METHOD objectIsValid
VAR_INPUT
	(* object which should be tested *)
	object	:CNM_AbstractObject.IObject;
	(* message if the assertion is false *)
	message	:AssertMessage;
END_VAR
IF (NOT THIS^.isObjectValid(object)) THEN
	THIS^.assertionWasWrong(message, THIS^.getDebugInfo('objectIsValid'));
END_IF
END_METHOD

(*

## Short summary
This assertion method checks if ``object``
precedes in sequence to ``objectToCompare``

.. <legal notes>

legal notes
=================
| SPDX-FileCopyrightText: © 2022 ekvip automation GmbH <info@ekvip.de>
| SPDX-License-Identifier: Apache-2.0
| For details check: Apache-2.0_

.. _Apache-2.0: https://www.apache.org/licenses/LICENSE-2.0

.. </legal notes>



*)

METHOD precedesInOrderTo
VAR_INPUT
	(* object which should be tested *)
	object			:CNM_AbstractObject.IObject;
	(* comparative object *)
	objectToCompare	:CNM_AbstractObject.IObject;
	(* message if the assertion is false *)
	message			:AssertMessage;
END_VAR
IF (THIS^.isObjectNull(THIS^.comperator)) THEN
	IF (THIS^.isObjectValid(object)) THEN
		IF (object.compareTo(objectToCompare) <> CNM_ReturnTypes.ComparationResult.SMALLER) THEN
			THIS^.assertionWasWrong(message, THIS^.getDebugInfo('precedesInOrderTo'));
		END_IF
	ELSIF (THIS^.isObjectValid(objectToCompare)) THEN
		IF (objectToCompare.compareTo(object) <= CNM_ReturnTypes.ComparationResult.EQUAL) THEN
			THIS^.assertionWasWrong(message, THIS^.getDebugInfo('precedesInOrderTo'));
		END_IF
	ELSE	
		THIS^.assertionWasWrong(message, THIS^.getDebugInfo('precedesInOrderTo'));
	END_IF
ELSIF (
	THIS^.comperator.compare(object, objectToCompare)
	<> CNM_ReturnTypes.ComparationResult.SMALLER
) THEN
	THIS^.assertionWasWrong(message, THIS^.getDebugInfo('precedesInOrderTo'));
END_IF
END_METHOD

(*

## Short summary
This allows you to set your own comperator for the methods
`IObjectAssertions.precedesInOrderTo`  
`IObjectAssertions.isEqualInOrderTo`  
`IObjectAssertions.isAfterInOrderTo`
to clear the comperator again, just call it with 0: ``foo.setComperator(comperator := 0);``

.. <legal notes>

legal notes
=================
| SPDX-FileCopyrightText: © 2022 ekvip automation GmbH <info@ekvip.de>
| SPDX-License-Identifier: Apache-2.0
| For details check: Apache-2.0_

.. _Apache-2.0: https://www.apache.org/licenses/LICENSE-2.0

.. </legal notes>



*)

METHOD setComperator
VAR_INPUT
	(* comperator to inject *)
	comperator	:CNM_AbstractObject.IComparator := 0;
END_VAR
THIS^.comperator := comperator;
END_METHOD

END_FUNCTION_BLOCK

// ---- Assertor/Assertions/PointerAssertions/classes/PointerAssertions.TcPOU
(*

## Short summary
This class provides assert statements for pointers  

.. <legal notes>

legal notes
=================
| SPDX-FileCopyrightText: © 2022 ekvip automation GmbH <info@ekvip.de>
| SPDX-License-Identifier: Apache-2.0
| For details check: Apache-2.0_

.. _Apache-2.0: https://www.apache.org/licenses/LICENSE-2.0

.. </legal notes>



*)

{attribute 'reflection'}
FUNCTION_BLOCK PointerAssertions EXTENDS AbstractAssertion IMPLEMENTS IPointerAssertions
VAR
END_VAR

(*

## Short summary
This abstract property returns the class name of the concrete object, 
It's for debugging purpose

.. <legal notes>

legal notes
=================
| SPDX-FileCopyrightText: © 2022 ekvip automation GmbH <info@ekvip.de>
| SPDX-License-Identifier: Apache-2.0
| For details check: Apache-2.0_

.. _Apache-2.0: https://www.apache.org/licenses/LICENSE-2.0

.. </legal notes>

*)

PROPERTY className :CNM_AbstractObject.ClassName
GET
className := 'CNM_Assertor.PointerAssertions';
END_GET
END_PROPERTY

(*

## Short summary
This assertion method checks if pointer is aligned with register size.

.. <legal notes>

legal notes
=================
| SPDX-FileCopyrightText: © 2025 ekvip automation GmbH <info@ekvip.de>
| SPDX-License-Identifier: Apache-2.0
| For details check: Apache-2.0_

.. _Apache-2.0: https://www.apache.org/licenses/LICENSE-2.0

.. </legal notes>



*)

METHOD isAligned
VAR_INPUT
	(* memory address *)
	address		:PVOID;
	(* message if the assertion is false *)
	message		:AssertMessage;
END_VAR
VAR CONSTANT
	SIZE :PVOID := SIZEOF(__XWORD);
END_VAR
IF (address MOD SIZE > 0) THEN
	THIS^.assertionWasWrong(message, THIS^.getDebugInfo('isAligned'));
END_IF
END_METHOD

(*

## Short summary
This assertion method checks if pointer is aligned with DWord size.

.. <legal notes>

legal notes
=================
| SPDX-FileCopyrightText: © 2025 ekvip automation GmbH <info@ekvip.de>
| SPDX-License-Identifier: Apache-2.0
| For details check: Apache-2.0_

.. _Apache-2.0: https://www.apache.org/licenses/LICENSE-2.0

.. </legal notes>



*)

METHOD isDwordAligned
VAR_INPUT
	(* memory address *)
	address		:PVOID;
	(* message if the assertion is false *)
	message		:AssertMessage;
END_VAR
VAR CONSTANT
	SIZE :PVOID := SIZEOF(DWORD);
END_VAR
IF (address MOD SIZE > 0) THEN
	THIS^.assertionWasWrong(message, THIS^.getDebugInfo('isAligned'));
END_IF
END_METHOD

(*

## Short summary
This assertion method checks if ``address1`` and ``address2`` refer to the same address

.. <legal notes>

legal notes
=================
| SPDX-FileCopyrightText: © 2022 ekvip automation GmbH <info@ekvip.de>
| SPDX-License-Identifier: Apache-2.0
| For details check: Apache-2.0_

.. _Apache-2.0: https://www.apache.org/licenses/LICENSE-2.0

.. </legal notes>



*)

METHOD isEqualTo
VAR_INPUT
	(* memory address *)
	address1	:PVOID;
	(* memory address *)
	address2	:PVOID;
	(* message if the assertion is false *)
	message		:AssertMessage;
END_VAR
IF (address1 <> address2) THEN
	THIS^.assertionWasWrong(message, THIS^.getDebugInfo('isEqualTo'));
END_IF
END_METHOD

(*

## Short summary
This assertion method checks if pointer is aligned with Lword size.

.. <legal notes>

legal notes
=================
| SPDX-FileCopyrightText: © 2025 ekvip automation GmbH <info@ekvip.de>
| SPDX-License-Identifier: Apache-2.0
| For details check: Apache-2.0_

.. _Apache-2.0: https://www.apache.org/licenses/LICENSE-2.0

.. </legal notes>



*)

METHOD isLwordAligned
VAR_INPUT
	(* memory address *)
	address		:PVOID;
	(* message if the assertion is false *)
	message		:AssertMessage;
END_VAR
VAR CONSTANT
	SIZE :PVOID := SIZEOF(LWORD);
END_VAR
IF (address MOD SIZE > 0) THEN
	THIS^.assertionWasWrong(message, THIS^.getDebugInfo('isAligned'));
END_IF
END_METHOD

(*

## Short summary
This assertion method checks if ``address1`` and ``address2`` refer not to the same address

.. <legal notes>

legal notes
=================
| SPDX-FileCopyrightText: © 2022 ekvip automation GmbH <info@ekvip.de>
| SPDX-License-Identifier: Apache-2.0
| For details check: Apache-2.0_

.. _Apache-2.0: https://www.apache.org/licenses/LICENSE-2.0

.. </legal notes>



*)

METHOD isNotEqualTo
VAR_INPUT
	(* memory address *)
	address1	:PVOID;
	(* memory address *)
	address2	:PVOID;
	(* message if the assertion is false *)
	message		:AssertMessage;
END_VAR
IF (address1 = address2) THEN
	THIS^.assertionWasWrong(message, THIS^.getDebugInfo('isNotEqualTo'));
END_IF
END_METHOD

(*

## Short summary
This assertion method checks if pointer is not null

.. <legal notes>

legal notes
=================
| SPDX-FileCopyrightText: © 2022 ekvip automation GmbH <info@ekvip.de>
| SPDX-License-Identifier: Apache-2.0
| For details check: Apache-2.0_

.. _Apache-2.0: https://www.apache.org/licenses/LICENSE-2.0

.. </legal notes>



*)

METHOD isNotNull
VAR_INPUT
	(* memory address *)
	address	:PVOID;
	(* message if the assertion is false *)
	message	:AssertMessage;
END_VAR
IF (address = 0) THEN
	THIS^.assertionWasWrong(message, THIS^.getDebugInfo('isNotNull'));
END_IF
END_METHOD

(*

## Short summary
This assertion method checks if memory areas are overlapping

.. <legal notes>

legal notes
=================
| SPDX-FileCopyrightText: © 2022 ekvip automation GmbH <info@ekvip.de>
| SPDX-License-Identifier: Apache-2.0
| For details check: Apache-2.0_

.. _Apache-2.0: https://www.apache.org/licenses/LICENSE-2.0

.. </legal notes>



*)

METHOD isNotOverlapping
VAR_INPUT
	(* memory address *)
	address1	:PVOID;
	(* memory address *)
	address2	:PVOID;
	(*the size of the memory area identified by address1*)
	sizeInBytes1		:UDINT;
	(*the size of the memory area identified by address2*)
	sizeInBytes2		:UDINT;
	(* message if the assertion is false *)
	message		:AssertMessage;
END_VAR
IF 	(( 
		address1 = address2
	) OR_ELSE(
		//address1 + sizeInBytes1 < address1 is to protect overflows caused by the calculation address1 + sizeInBytes1
		(address1 < address2) AND_THEN ((address1 + sizeInBytes1 < address1) OR_ELSE ((address1 + sizeInBytes1) >= address2))
	) OR_ELSE (
		//address2 + sizeInBytes2 < address2 is to protect overflows caused by the calculation address2 + sizeInBytes2
		(address1 > address2) AND_THEN (((address2 + sizeInBytes2 < address2) OR_ELSE ((address2 + sizeInBytes2) >= address1)))
	)
) THEN
		THIS^.assertionWasWrong(message, THIS^.getDebugInfo('isNotOverlapping'));
END_IF
END_METHOD

(*

## Short summary
This assertion method checks if pointer is null

.. <legal notes>

legal notes
=================
| SPDX-FileCopyrightText: © 2022 ekvip automation GmbH <info@ekvip.de>
| SPDX-License-Identifier: Apache-2.0
| For details check: Apache-2.0_

.. _Apache-2.0: https://www.apache.org/licenses/LICENSE-2.0

.. </legal notes>



*)

METHOD isNull
VAR_INPUT
	(* memory address *)
	address	:PVOID;
	(* message if the assertion is false *)
	message	:AssertMessage;
END_VAR
IF (address <> 0) THEN
	THIS^.assertionWasWrong(message, THIS^.getDebugInfo('isNull'));
END_IF
END_METHOD

(*

## Short summary
This assertion method checks if memory areas are overlapping

.. <legal notes>

legal notes
=================
| SPDX-FileCopyrightText: © 2022 ekvip automation GmbH <info@ekvip.de>
| SPDX-License-Identifier: Apache-2.0
| For details check: Apache-2.0_

.. _Apache-2.0: https://www.apache.org/licenses/LICENSE-2.0

.. </legal notes>



*)

METHOD isOverlapping
VAR_INPUT
	(* memory address *)
	address1	:PVOID;
	(* memory address *)
	address2	:PVOID;
	(*the size of the memory area identified by address1*)
	sizeInBytes1		:UDINT;
	(*the size of the memory area identified by address2*)
	sizeInBytes2		:UDINT;
	(* message if the assertion is false *)
	message		:AssertMessage;
END_VAR
RETURN(address1 = address2);
IF ((
		(address1 < address2) AND_THEN ((address1 + sizeInBytes1) < address2)
	) OR_ELSE (
		(address1 > address2) AND_THEN ((address2 + sizeInBytes2) < address1)
	)
) THEN
	THIS^.assertionWasWrong(message, THIS^.getDebugInfo('isOverlapping'));
END_IF;
END_METHOD

(*

## Short summary
This assertion method checks if pointer is valid.
That means the pointer and size are not zero,
the pointer is in a valid area.

**Attention:** 
	Validity of the pointer will be proofed for 32 bit systems only.
	For other systems it's an optimistic estimate.

.. <legal notes>

legal notes
=================
| SPDX-FileCopyrightText: © 2022 ekvip automation GmbH <info@ekvip.de>
| SPDX-License-Identifier: Apache-2.0
| For details check: Apache-2.0_

.. _Apache-2.0: https://www.apache.org/licenses/LICENSE-2.0

.. </legal notes>



*)

METHOD isValid
VAR_INPUT
	(* memory address *)
	address		:PVOID;
	(* number of bytes *)
	sizeInBytes	:UDINT;
	(* message if the assertion is false *)
	message		:AssertMessage;
END_VAR
VAR
	{attribute 'displaymode':='hex'}
	stackAddress	:__XWORD;
	testPointer		:POINTER TO BYTE := NULL;
	testByte		:BYTE;
	exc				: __SYSTEM.ExceptionCode;
END_VAR
VAR CONSTANT
	{attribute 'displaymode':='hex'}
	NULL :__XWORD := 0;
	{attribute 'displaymode':='hex'}
	REGISTER_SIZE :UDINT := SIZEOF(__XWORD);
	(* 0x400000 is 4096kb and this is the max configurable stack size *)
	{attribute 'displaymode':='hex'}
	MAX_STACK_SIZE :__XWORD := 16#0040_0000;
END_VAR
stackAddress := ADR(stackAddress);
IF (
	(address = NULL) 
	OR_ELSE (sizeInBytes = NULL)
	//check for overflow
	OR_ELSE (address + sizeInBytes < address)
	OR_ELSE (
		(Tc2_System.F_CheckMemoryArea(pData := address, nSize := sizeInBytes) = Tc2_System.E_TcMemoryArea.Unknown)
		AND_THEN (address < ABS(stackAddress - MAX_STACK_SIZE))
	)
) THEN
	THIS^.assertionWasWrong(message, THIS^.getDebugInfo('isValid'));
ELSE
	testPointer := address;
	__TRY
		testByte := testPointer^;
	__CATCH(exc)
		THIS^.assertionWasWrong(message, THIS^.getDebugInfo('isValid'));
	__ENDTRY
END_IF
END_METHOD

(*

## Short summary
This assertion method checks if pointer is aligned with word size.

.. <legal notes>

legal notes
=================
| SPDX-FileCopyrightText: © 2025 ekvip automation GmbH <info@ekvip.de>
| SPDX-License-Identifier: Apache-2.0
| For details check: Apache-2.0_

.. _Apache-2.0: https://www.apache.org/licenses/LICENSE-2.0

.. </legal notes>



*)

METHOD isWordAligned
VAR_INPUT
	(* memory address *)
	address		:PVOID;
	(* message if the assertion is false *)
	message		:AssertMessage;
END_VAR
VAR CONSTANT
	SIZE :PVOID := SIZEOF(WORD);
END_VAR
IF (address MOD SIZE > 0) THEN
	THIS^.assertionWasWrong(message, THIS^.getDebugInfo('isAligned'));
END_IF
END_METHOD

(*

## Short summary
This assertion method checks if pointer refers to cnc area

.. <legal notes>

legal notes
=================
| SPDX-FileCopyrightText: © 2022 ekvip automation GmbH <info@ekvip.de>
| SPDX-License-Identifier: Apache-2.0
| For details check: Apache-2.0_

.. _Apache-2.0: https://www.apache.org/licenses/LICENSE-2.0

.. </legal notes>



*)

METHOD memoryAreaIsCnc
VAR_INPUT
	(* memory address *)
	address		:PVOID;
	(* number of bytes *)
	sizeInBytes	:UDINT;
	(* message if the assertion is false *)
	message		:AssertMessage;
END_VAR
IF (
	Tc2_System.F_CheckMemoryArea(
		pData := address,
		nSize := sizeInBytes
	) <> Tc2_System.E_TcMemoryArea.CNC
) THEN
	THIS^.assertionWasWrong(message, THIS^.getDebugInfo('memoryAreaIsCnc'));
END_IF
END_METHOD

(*

## Short summary
This assertion method checks if pointer refers to dynamic area

.. <legal notes>

legal notes
=================
| SPDX-FileCopyrightText: © 2022 ekvip automation GmbH <info@ekvip.de>
| SPDX-License-Identifier: Apache-2.0
| For details check: Apache-2.0_

.. _Apache-2.0: https://www.apache.org/licenses/LICENSE-2.0

.. </legal notes>



*)

METHOD memoryAreaIsDynamic
VAR_INPUT
	(* memory address *)
	address		:PVOID;
	(* number of bytes *)
	sizeInBytes	:UDINT;
	(* message if the assertion is false *)
	message		:AssertMessage;
END_VAR
IF (
	Tc2_System.F_CheckMemoryArea(
		pData := address,
		nSize := sizeInBytes
	) <> Tc2_System.E_TcMemoryArea.Dynamic
) THEN
	THIS^.assertionWasWrong(message, THIS^.getDebugInfo('memoryAreaIsDynamic'));
END_IF
END_METHOD

(*

## Short summary
This assertion method checks if pointer refers not to cnc area

.. <legal notes>

legal notes
=================
| SPDX-FileCopyrightText: © 2022 ekvip automation GmbH <info@ekvip.de>
| SPDX-License-Identifier: Apache-2.0
| For details check: Apache-2.0_

.. _Apache-2.0: https://www.apache.org/licenses/LICENSE-2.0

.. </legal notes>



*)

METHOD memoryAreaIsNotCnc
VAR_INPUT
	(* memory address *)
	address		:PVOID;
	(* number of bytes *)
	sizeInBytes	:UDINT;
	(* message if the assertion is false *)
	message		:AssertMessage;
END_VAR
IF (
	Tc2_System.F_CheckMemoryArea(
		pData := address,
		nSize := sizeInBytes
	) = Tc2_System.E_TcMemoryArea.CNC
) THEN
	THIS^.assertionWasWrong(message, THIS^.getDebugInfo('memoryAreaIsNotCnc'));
END_IF
END_METHOD

(*

## Short summary
This assertion method checks if pointer refers not to dynamic area

.. <legal notes>

legal notes
=================
| SPDX-FileCopyrightText: © 2022 ekvip automation GmbH <info@ekvip.de>
| SPDX-License-Identifier: Apache-2.0
| For details check: Apache-2.0_

.. _Apache-2.0: https://www.apache.org/licenses/LICENSE-2.0

.. </legal notes>



*)

METHOD memoryAreaIsNotDynamic
VAR_INPUT
	(* memory address *)
	address		:PVOID;
	(* number of bytes *)
	sizeInBytes	:UDINT;
	(* message if the assertion is false *)
	message		:AssertMessage;
END_VAR
IF (
	Tc2_System.F_CheckMemoryArea(
		pData := address,
		nSize := sizeInBytes
	) = Tc2_System.E_TcMemoryArea.Dynamic
) THEN
	THIS^.assertionWasWrong(message, THIS^.getDebugInfo('memoryAreaIsNotDynamic'));
END_IF
END_METHOD

(*

## Short summary
This assertion method checks if pointer refers not to static area

.. <legal notes>

legal notes
=================
| SPDX-FileCopyrightText: © 2022 ekvip automation GmbH <info@ekvip.de>
| SPDX-License-Identifier: Apache-2.0
| For details check: Apache-2.0_

.. _Apache-2.0: https://www.apache.org/licenses/LICENSE-2.0

.. </legal notes>



*)

METHOD memoryAreaIsNotStatic
VAR_INPUT
	(* memory address *)
	address		:PVOID;
	(* number of bytes *)
	sizeInBytes	:UDINT;
	(* message if the assertion is false *)
	message		:AssertMessage;
END_VAR
IF (
	Tc2_System.F_CheckMemoryArea(
		pData := address,
		nSize := sizeInBytes
	) = Tc2_System.E_TcMemoryArea.Static
) THEN
	THIS^.assertionWasWrong(message, THIS^.getDebugInfo('memoryAreaIsNotStatic'));
END_IF
END_METHOD

(*

## Short summary
This assertion method checks if pointer is not at memory area unknown

.. <legal notes>

legal notes
=================
| SPDX-FileCopyrightText: © 2022 ekvip automation GmbH <info@ekvip.de>
| SPDX-License-Identifier: Apache-2.0
| For details check: Apache-2.0_

.. _Apache-2.0: https://www.apache.org/licenses/LICENSE-2.0

.. </legal notes>



*)

METHOD memoryAreaIsNotUnkown
VAR_INPUT
	(* memory address *)
	address		:PVOID;
	(* number of bytes *)
	sizeInBytes	:UDINT;
	(* message if the assertion is false *)
	message		:AssertMessage;
END_VAR
IF (
	Tc2_System.F_CheckMemoryArea(
		pData := address,
		nSize := sizeInBytes
	) = Tc2_System.E_TcMemoryArea.Unknown
) THEN
	THIS^.assertionWasWrong(message, THIS^.getDebugInfo('memoryAreaIsNotUnkown'));
END_IF
END_METHOD

(*

## Short summary
This assertion method checks if pointer refers to static area

.. <legal notes>

legal notes
=================
| SPDX-FileCopyrightText: © 2022 ekvip automation GmbH <info@ekvip.de>
| SPDX-License-Identifier: Apache-2.0
| For details check: Apache-2.0_

.. _Apache-2.0: https://www.apache.org/licenses/LICENSE-2.0

.. </legal notes>



*)

METHOD memoryAreaIsStatic
VAR_INPUT
	(* memory address *)
	address		:PVOID;
	(* number of bytes *)
	sizeInBytes	:UDINT;
	(* message if the assertion is false *)
	message		:AssertMessage;
END_VAR
IF (
	Tc2_System.F_CheckMemoryArea(
		pData := address,
		nSize := sizeInBytes
	) <> Tc2_System.E_TcMemoryArea.Static
) THEN
	THIS^.assertionWasWrong(message, THIS^.getDebugInfo('memoryAreaIsStatic'));
END_IF
END_METHOD

(*

## Short summary
This assertion method checks if pointer refers not to an unknown area

.. <legal notes>

legal notes
=================
| SPDX-FileCopyrightText: © 2022 ekvip automation GmbH <info@ekvip.de>
| SPDX-License-Identifier: Apache-2.0
| For details check: Apache-2.0_

.. _Apache-2.0: https://www.apache.org/licenses/LICENSE-2.0

.. </legal notes>



*)

METHOD memoryAreaIsUnkown
VAR_INPUT
	(* memory address *)
	address		:PVOID;
	(* number of bytes *)
	sizeInBytes	:UDINT;
	(* message if the assertion is false *)
	message		:AssertMessage;
END_VAR
IF (
	Tc2_System.F_CheckMemoryArea(
		pData := address,
		nSize := sizeInBytes
	) <> Tc2_System.E_TcMemoryArea.Unknown
) THEN
	THIS^.assertionWasWrong(message, THIS^.getDebugInfo('memoryAreaIsUnkown'));
END_IF
END_METHOD

END_FUNCTION_BLOCK

// ---- Assertor/Assertions/StringAssertion/classes/StringAssertions.TcPOU
(*

## Short summary

This class provides assert statements for strings
For UTF-16 strings up to 255 ``WORD`` (``WSTRING(Tc2_System.MAX_STRING_LENGTH)``) use the property `IStringAssertions.utf16`.
For windows-1252 strings up to 255 ``BYTE`` (``Tc2_System.T_MaxString``) use the property `IStringAssertions.windows1252`.
For windows-1252 or UTF-16 strings that are longer, use the property `IStringAssertions.anyString`  

.. <legal notes>

legal notes
=================
| SPDX-FileCopyrightText: © 2022 ekvip automation GmbH <info@ekvip.de>
| SPDX-License-Identifier: Apache-2.0
| For details check: Apache-2.0_

.. _Apache-2.0: https://www.apache.org/licenses/LICENSE-2.0

.. </legal notes>



*)

{attribute 'reflection'}
FUNCTION_BLOCK INTERNAL StringAssertions EXTENDS CNM_AbstractObject.Object IMPLEMENTS IStringAssertions, IAssertCallBackSetter
VAR
	(* class to handle windows-1252 and windows-1251 assertions *)
	win125xStringAssertions	:Windows125xStringAssertions();
	(* class to handle UTF-16 assertions *)
	utf16StringAssertions	:Utf16StringAssertions();
	(* class to handle UTF-8 assertions *)
	utf8StringAssertions	:Utf8StringAssertions();
	(* class to handle Unicode assertions with anys string*)
	UnicodeAssertions :UnicodeAssertions();
END_VAR

(*

## Short summary
This abstract property returns the class name of the concrete object, 
It's for debugging purpose

.. <legal notes>

legal notes
=================
| SPDX-FileCopyrightText: © 2022 ekvip automation GmbH <info@ekvip.de>
| SPDX-License-Identifier: Apache-2.0
| For details check: Apache-2.0_

.. _Apache-2.0: https://www.apache.org/licenses/LICENSE-2.0

.. </legal notes>

*)

PROPERTY className :CNM_AbstractObject.ClassName
GET
className := 'CNM_Assertor.StringAssertions';
END_GET
END_PROPERTY

(*

## Short summary
This methods is the setter for the callback class if an assertion was false

.. <legal notes>

legal notes
=================
| SPDX-FileCopyrightText: © 2022 ekvip automation GmbH <info@ekvip.de>
| SPDX-License-Identifier: Apache-2.0
| For details check: Apache-2.0_

.. _Apache-2.0: https://www.apache.org/licenses/LICENSE-2.0

.. </legal notes>



*)

METHOD setCallBack
VAR_INPUT
	(* the class that must be informed if an assertion is false *)
	callBack	: IAssertCallBack;
END_VAR
THIS^.utf16StringAssertions.setCallBack(callBack);
THIS^.win125xStringAssertions.setCallBack(callBack);
THIS^.utf8StringAssertions.setCallBack(callBack);
THIS^.UnicodeAssertions.setCallBack(callBack);
END_METHOD

(*

## Short summary
Returns an interface `IUnicodeStringAssertions` with assert statements,
for UTF-8 and UTF-16 strings with an undefined length.

**Attention:** 
	All strings are handled as null terminated byte/word streams.
	For UTF-8 is end of the string 16#00
	For UTF-16 is end of the string 16#00_00

**Attention:** 
	The interface `IUnicodeAssertions` uses ``ANY_STRING``, 
	for this it's not possible to use literals/constants,
	because for ``ANY`` types generates the compiler ``__SYSTEM.AnyType``
	and ``__SYSTEM.AnyType`` contains a pointer  

.. <legal notes>

legal notes
=================
| SPDX-FileCopyrightText: © 2022 ekvip automation GmbH <info@ekvip.de>
| SPDX-License-Identifier: Apache-2.0
| For details check: Apache-2.0_

.. _Apache-2.0: https://www.apache.org/licenses/LICENSE-2.0

.. </legal notes>

*)
PROPERTY unicode :IUnicodeStringAssertions
GET
unicode := THIS^.UnicodeAssertions;
END_GET
END_PROPERTY

(*

## Short summary
Returns an interface `IUtf16StringAssertions` with assert statements
for UTF-16 strings until 255 ``WORD`` length (``WSTRING(Tc2_System.MAX_STRING_LENGTH)``)

.. <legal notes>

legal notes
=================
| SPDX-FileCopyrightText: © 2022 ekvip automation GmbH <info@ekvip.de>
| SPDX-License-Identifier: Apache-2.0
| For details check: Apache-2.0_

.. _Apache-2.0: https://www.apache.org/licenses/LICENSE-2.0

.. </legal notes>

*)

PROPERTY utf16 :IUtf16StringAssertions
GET
utf16 := THIS^.utf16StringAssertions;
END_GET
END_PROPERTY

(*

## Short summary
Returns an interface `IUtf8StringAssertions` with assert statements
for UTF-8 strings up to 255 bytes length (``STRING(Tc2_System.MAX_STRING_LENGTH)``)

.. <legal notes>

legal notes
=================
| SPDX-FileCopyrightText: © 2022 ekvip automation GmbH <info@ekvip.de>
| SPDX-License-Identifier: Apache-2.0
| For details check: Apache-2.0_

.. _Apache-2.0: https://www.apache.org/licenses/LICENSE-2.0

.. </legal notes>

*)

PROPERTY utf8 :IUtf8StringAssertions
GET
utf8 := THIS^.utf8StringAssertions;
END_GET
END_PROPERTY

(*

## Short summary
Returns an interface `IWindows125xStringAssertions` with assert statements for 8-bit 
windows-1252 and windows-1251 strings up to 255 characters length (``Tc2_System.T_MaxString``).
Use Tc2_Utilities.GLOBAL_SBCS_TABLE variable to select required encoding

.. <legal notes>

legal notes
=================
| SPDX-FileCopyrightText: © 2022 ekvip automation GmbH <info@ekvip.de>
| SPDX-License-Identifier: Apache-2.0
| For details check: Apache-2.0_

.. _Apache-2.0: https://www.apache.org/licenses/LICENSE-2.0

.. </legal notes>

*)

PROPERTY windows125x :IWindows125xStringAssertions
GET
windows125x := THIS^.win125xStringAssertions;
END_GET
END_PROPERTY

END_FUNCTION_BLOCK

// ---- Assertor/Assertions/StringAssertion/Win125x/classes/Windows125xStringAssertions.TcPOU
(*

## Short summary
This class provides assert statements for Windows-1252 and Windows-1251 strings up to 255 characters length. 
Used encoding is specified in ``Tc2_Utilities.GLOBAL_SBCS_TABLE`` global variable

**Attention:** 
	All strings are handled as null-terminated byte streams

.. <legal notes>

legal notes
=================
| SPDX-FileCopyrightText: © 2024 ekvip automation GmbH <info@ekvip.de>
| SPDX-License-Identifier: Apache-2.0
| For details check: Apache-2.0_

.. _Apache-2.0: https://www.apache.org/licenses/LICENSE-2.0

.. </legal notes>



*)

{attribute 'reflection'}
FUNCTION_BLOCK INTERNAL Windows125xStringAssertions EXTENDS AbstractAssertion IMPLEMENTS IWindows125xStringAssertions
VAR
	(* class to handle the windows-1252 and windows-1251 string assertions *)  
	assertion	:Windows125xStringPointerAssertions();
END_VAR

(*

## Short summary
This abstract property returns the class name of the concrete object, 
It's for debugging purpose

.. <legal notes>

legal notes
=================
| SPDX-FileCopyrightText: © 2022 ekvip automation GmbH <info@ekvip.de>
| SPDX-License-Identifier: Apache-2.0
| For details check: Apache-2.0_

.. _Apache-2.0: https://www.apache.org/licenses/LICENSE-2.0

.. </legal notes>

*)

PROPERTY className :CNM_AbstractObject.ClassName
GET
className := 'CNM_Assertor.Windows125xStringAssertions';
END_GET
END_PROPERTY

(*

## Short summary
This assertion method checks if the current string ``stringToCheck`` contains the search string ``searchString``.
Processed strings must be in UTF-8 encoding

.. <legal notes>

legal notes
=================
| SPDX-FileCopyrightText: © 2024 ekvip automation GmbH <info@ekvip.de>
| SPDX-License-Identifier: Apache-2.0
| For details check: Apache-2.0_

.. _Apache-2.0: https://www.apache.org/licenses/LICENSE-2.0

.. </legal notes>



*)

METHOD contains
VAR_INPUT
	(* current string to check *)
	stringToCheck	:Tc2_System.T_MaxString;
	(* string must be found in ``stringToCheck`` *)
	searchString	:Tc2_System.T_MaxString;
	(* message if the assertion is false *)
	message			:AssertMessage;
	(* used Single Byte Character Set (SBCS), is set in Tc2_Utilities.GLOBAL_SBCS_TABLE *)
	sbcsType 		:Tc2_Utilities.E_SBCSType := Tc2_Utilities.E_SBCSType.eSBCS_WesternEuropean;
	(* ``TRUE`` means ignore cases; ``FALSE`` means that cases must be equal too *)
	ignoreCases		:BOOL := FALSE;
END_VAR
assertion.contains(
	stringToCheck 	:= ADR(stringToCheck),
	searchString  	:= ADR(searchString),
	ignoreCases 	:= ignoreCases,
	message 		:= message,
	sbcsType 		:= sbcsType
);
END_METHOD

(*

## Short summary
This assertion method checks if the current string ``stringToCheck`` doesn't contain the search string ``searchString``.
Processed strings must be in UTF-8 encoding

.. <legal notes>

legal notes
=================
| SPDX-FileCopyrightText: © 2024 ekvip automation GmbH <info@ekvip.de>
| SPDX-License-Identifier: Apache-2.0
| For details check: Apache-2.0_

.. _Apache-2.0: https://www.apache.org/licenses/LICENSE-2.0

.. </legal notes>



*)

METHOD containsNo
VAR_INPUT
	(* current string to check *)
	stringToCheck	:Tc2_System.T_MaxString;
	(* string that must not be found in ``stringToCheck`` *)
	searchString	:Tc2_System.T_MaxString;
	(* message if the assertion is false *)
	message			:AssertMessage;
	(* used Single Byte Character Set (SBCS), is set in Tc2_Utilities.GLOBAL_SBCS_TABLE *)
	sbcsType 		:Tc2_Utilities.E_SBCSType := Tc2_Utilities.E_SBCSType.eSBCS_WesternEuropean;
	(* ``TRUE`` means ignore cases; ``FALSE`` means that cases must be equal too *)
	ignoreCases		:BOOL := FALSE;
END_VAR
THIS^.assertion.containsNo(
	stringToCheck 	:= ADR(stringToCheck),
	searchString 	:= ADR(searchString),
	ignoreCases 	:= ignoreCases,
	message 		:= message,
	sbcsType 		:= sbcsType
);
END_METHOD

(*

## Short summary
This assertion method checks if the current string ``stringToCheck`` ends with the string ``end``.
Processed strings must be in UTF-8 encoding

.. <legal notes>

legal notes
=================
| SPDX-FileCopyrightText: © 2024 ekvip automation GmbH <info@ekvip.de>
| SPDX-License-Identifier: Apache-2.0
| For details check: Apache-2.0_

.. _Apache-2.0: https://www.apache.org/licenses/LICENSE-2.0

.. </legal notes>



*)

METHOD endsWith
VAR_INPUT
	(* current string to check *)
	stringToCheck	:Tc2_System.T_MaxString;
	(* expected end of ``stringToCheck`` *)
	end				:Tc2_System.T_MaxString;
	(* message if the assertion is false *)
	message			:AssertMessage;
	(* used Single Byte Character Set (SBCS), is set in Tc2_Utilities.GLOBAL_SBCS_TABLE *)
	sbcsType 		:Tc2_Utilities.E_SBCSType := Tc2_Utilities.E_SBCSType.eSBCS_WesternEuropean;
	(* ``TRUE`` means ignore cases; ``FALSE`` means that cases must be equal too *)
	ignoreCases		:BOOL := FALSE;
	(* ``TRUE`` means truncation of spaces on the right side of ``stringToCheck``*)
	trim		:BOOL := FALSE;
END_VAR
assertion.endsWith(
	stringToCheck	:= ADR(stringToCheck),
	end				:= ADR(end),
	ignoreCases		:= ignoreCases,
	trim			:= trim,
	message			:= message,
	sbcsType 		:= sbcsType
);
END_METHOD

(*

## Short summary
This assertion method checks if the current string ``stringToCheck`` is empty.
Processed strings must be in UTF-8 encoding

.. <legal notes>

legal notes
=================
| SPDX-FileCopyrightText: © 2024 ekvip automation GmbH <info@ekvip.de>
| SPDX-License-Identifier: Apache-2.0
| For details check: Apache-2.0_

.. _Apache-2.0: https://www.apache.org/licenses/LICENSE-2.0

.. </legal notes>



*)

METHOD isEmpty
VAR_INPUT
	(* current string to check *)
	stringToCheck	:Tc2_System.T_MaxString;
	(* message if the assertion is false *)
	message			:AssertMessage;
END_VAR
IF (stringToCheck <> '') THEN
	THIS^.assertionWasWrong(message, THIS^.getDebugInfo('isEmpty'));
END_IF
END_METHOD

(*

## Short summary
This assertion method checks if the current string ``stringToCheck`` is equal to ``expected``.
Processed strings must be in UTF-8 encoding

.. <legal notes>

legal notes
=================
| SPDX-FileCopyrightText: © 2024 ekvip automation GmbH <info@ekvip.de>
| SPDX-License-Identifier: Apache-2.0
| For details check: Apache-2.0_

.. _Apache-2.0: https://www.apache.org/licenses/LICENSE-2.0

.. </legal notes>



*)

METHOD isEqualTo
VAR_INPUT
	(* current string to check *)
	stringToCheck	:Tc2_System.T_MaxString;
	(* ``stringToCheck`` must be equal to expected *)
	expected		:Tc2_System.T_MaxString;
	(* message if the assertion is false *)
	message			:AssertMessage;
	(* used Single Byte Character Set (SBCS), is set in Tc2_Utilities.GLOBAL_SBCS_TABLE *)
	sbcsType 		:Tc2_Utilities.E_SBCSType := Tc2_Utilities.E_SBCSType.eSBCS_WesternEuropean;
	(* ``TRUE`` means ignore cases; ``FALSE`` means that cases must be equal too *)
	ignoreCases		:BOOL := FALSE;
END_VAR
assertion.isEqualTo(
	stringToCheck	:= ADR(stringToCheck),
	expected		:= ADR(expected),
	ignoreCases		:= ignoreCases,
	message			:= message,
	sbcsType 		:= sbcsType
);
END_METHOD

(*

## Short summary
This assertion method checks if the current string ``stringToCheck`` is not empty.
Processed strings must be in UTF-8 encoding

.. <legal notes>

legal notes
=================
| SPDX-FileCopyrightText: © 2024 ekvip automation GmbH <info@ekvip.de>
| SPDX-License-Identifier: Apache-2.0
| For details check: Apache-2.0_

.. _Apache-2.0: https://www.apache.org/licenses/LICENSE-2.0

.. </legal notes>



*)

METHOD isNotEmpty
VAR_INPUT
	(* current string to check *)
	stringToCheck	:Tc2_System.T_MaxString;
	(* message if the assertion is false *)
	message			:AssertMessage;
END_VAR
IF (stringToCheck = '') THEN
	THIS^.assertionWasWrong(message, THIS^.getDebugInfo('isEmpty'));
END_IF
END_METHOD

(*

## Short summary
This assertion method checks if the current string ``stringToCheck`` is not equal to ``unexpected``.
Processed strings must be in UTF-8 encoding

.. <legal notes>

legal notes
=================
| SPDX-FileCopyrightText: © 2024 ekvip automation GmbH <info@ekvip.de>
| SPDX-License-Identifier: Apache-2.0
| For details check: Apache-2.0_

.. _Apache-2.0: https://www.apache.org/licenses/LICENSE-2.0

.. </legal notes>



*)

METHOD isNotEqualTo
VAR_INPUT
	(* current string to check *)
	stringToCheck	:Tc2_System.T_MaxString;
	(* ``stringToCheck`` must be not equal to expected *)
	unexpected		:Tc2_System.T_MaxString;
	(* message if the assertion is false *)
	message			:AssertMessage;
	(* used Single Byte Character Set (SBCS), is set in Tc2_Utilities.GLOBAL_SBCS_TABLE *)
	sbcsType 		:Tc2_Utilities.E_SBCSType := Tc2_Utilities.E_SBCSType.eSBCS_WesternEuropean;
	(* ``TRUE`` means ignore cases; ``FALSE`` means that cases must be equal too *)
	ignoreCases		:BOOL := FALSE;
END_VAR
THIS^.assertion.isNotEqualTo(
	stringToCheck	:= ADR(stringToCheck),
	unexpected		:= ADR(unexpected),
	ignoreCases		:= ignoreCases,
	message			:= message,
	sbcsType 		:= sbcsType
);
END_METHOD

(*

## Short summary
This assertion method checks if the current string ``stringToCheck`` length is between ``minLength`` and ``maxLength``.
Processed strings must be in UTF-8 encoding

.. <legal notes>

legal notes
=================
| SPDX-FileCopyrightText: © 2024 ekvip automation GmbH <info@ekvip.de>
| SPDX-License-Identifier: Apache-2.0
| For details check: Apache-2.0_

.. _Apache-2.0: https://www.apache.org/licenses/LICENSE-2.0

.. </legal notes>



*)

METHOD lengthIsBetween
VAR_INPUT
	(* current string to check *)
	stringToCheck	:Tc2_System.T_MaxString;
	(* lower limit of the string length *)
	minLength		:USINT;
	(* upper limit of the string length *)
	maxLength		:USINT;
	(* message if the assertion is false *)
	message			:AssertMessage;
END_VAR
THIS^.assertion.lengthIsBetween(
	stringToCheck	:= ADR(stringToCheck),
	minLength		:= minLength,
	maxLength		:= maxLength,
	message			:= message
);
END_METHOD

(*

## Short summary
This assertion method checks if the current string ``stringToCheck`` length is equal to ``expectedLength``.
Processed strings must be in UTF-8 encoding

.. <legal notes>

legal notes
=================
| SPDX-FileCopyrightText: © 2024 ekvip automation GmbH <info@ekvip.de>
| SPDX-License-Identifier: Apache-2.0
| For details check: Apache-2.0_

.. _Apache-2.0: https://www.apache.org/licenses/LICENSE-2.0

.. </legal notes>



*)

METHOD lengthIsExact
VAR_INPUT
	(* current string to check *)
	stringToCheck	:Tc2_System.T_MaxString;
	(* expected length of ``stringToCheck`` *)
	expectedLength	:USINT;
	(* message if the assertion is false *)
	message			:AssertMessage;
END_VAR
THIS^.assertion.lengthIsExact(
	stringToCheck	:= ADR(stringToCheck),
	expectedLength	:= expectedLength,
	message			:= message
);
END_METHOD

(*

## Short summary
This assertion method checks if the current string ``stringToCheck`` length is equal or less than to ``maxLength``.
Processed strings must be in UTF-8 encoding

.. <legal notes>

legal notes
=================
| SPDX-FileCopyrightText: © 2024 ekvip automation GmbH <info@ekvip.de>
| SPDX-License-Identifier: Apache-2.0
| For details check: Apache-2.0_

.. _Apache-2.0: https://www.apache.org/licenses/LICENSE-2.0

.. </legal notes>



*)

METHOD lengthIsMax
VAR_INPUT
	(* current string to check *)
	stringToCheck	:Tc2_System.T_MaxString;
	(* upper limit of the length of ``stringToCheck`` *)
	maxLength		:USINT;
	(* message if the assertion is false *)
	message			:AssertMessage;
END_VAR
THIS^.assertion.lengthIsMax(
	stringToCheck	:= ADR(stringToCheck),
	maxLength		:= maxLength,
	message			:= message
);
END_METHOD

(*

## Short summary
This assertion method checks if the current string ``stringToCheck`` length is equal or grater than to ``minLength``.
Processed strings must be in UTF-8 encoding

.. <legal notes>

legal notes
=================
| SPDX-FileCopyrightText: © 2024 ekvip automation GmbH <info@ekvip.de>
| SPDX-License-Identifier: Apache-2.0
| For details check: Apache-2.0_

.. _Apache-2.0: https://www.apache.org/licenses/LICENSE-2.0

.. </legal notes>



*)

METHOD lengthIsMin
VAR_INPUT
	(* current string to check *)
	stringToCheck	:Tc2_System.T_MaxString;
	(* lower limit of the length of ``stringToCheck`` *)
	minLength		:USINT;
	(* message if the assertion is false *)
	message			:AssertMessage;
END_VAR
THIS^.assertion.lengthIsMin(
	stringToCheck	:= ADR(stringToCheck),
	minLength		:= minLength,
	message			:= message
);
END_METHOD

(*

## Short summary
This methods is the setter for the callback class if an assertion was false

.. <legal notes>

legal notes
=================
| SPDX-FileCopyrightText: © 2024 ekvip automation GmbH <info@ekvip.de>
| SPDX-License-Identifier: Apache-2.0
| For details check: Apache-2.0_

.. _Apache-2.0: https://www.apache.org/licenses/LICENSE-2.0

.. </legal notes>



*)

METHOD setCallBack
VAR_INPUT
	(* the class that must be informed if an assertion is false *)
	callBack	:IAssertCallBack;  
END_VAR
SUPER^.setCallBack(callBack);
THIS^.assertion.setCallBack(callBack);
END_METHOD

(*

## Short summary
This assertion method checks if the current string ``stringToCheck`` starts with string ``start``.
Processed strings must be in UTF-8 encoding

.. <legal notes>

legal notes
=================
| SPDX-FileCopyrightText: © 2024 ekvip automation GmbH <info@ekvip.de>
| SPDX-License-Identifier: Apache-2.0
| For details check: Apache-2.0_

.. _Apache-2.0: https://www.apache.org/licenses/LICENSE-2.0

.. </legal notes>



*)

METHOD startsWith
VAR_INPUT
	(* current string to check *)
	stringToCheck	:Tc2_System.T_MaxString;
	(* expected start of ``stringToCheck`` *)
	start			:Tc2_System.T_MaxString;
	(* message if the assertion is false *)
	message			:AssertMessage;
	(* used Single Byte Character Set (SBCS), is set in Tc2_Utilities.GLOBAL_SBCS_TABLE *)
	sbcsType 		:Tc2_Utilities.E_SBCSType := Tc2_Utilities.E_SBCSType.eSBCS_WesternEuropean;
	(* ``TRUE`` means ignore cases; ``FALSE`` means that cases must be equal too *)
	ignoreCases		:BOOL := FALSE;
	(* ``TRUE`` means truncation of spaces on the left side of ``stringToCheck``*)
	trim		:BOOL := FALSE;
END_VAR
assertion.startsWith(
	stringToCheck	:= ADR(stringToCheck),
	start			:= ADR(start),
	ignoreCases		:= ignoreCases,
	trim			:= trim,
	message			:= message,
	sbcsType 		:= sbcsType
);
END_METHOD

END_FUNCTION_BLOCK

// ---- Assertor/Assertions/StringAssertion/Win125x/classes/Windows125xStringPointerAssertions.TcPOU
(*

## Short summary
This class provides assert statements for Windows-1252 and Windows-1251 strings.
Used encoding is specified in ``Tc2_Utilities.GLOBAL_SBCS_TABLE`` global variable

**Attention:** 
	All strings are handled as null-terminated byte streams

.. <legal notes>

legal notes
=================
| SPDX-FileCopyrightText: © 2024 ekvip automation GmbH <info@ekvip.de>
| SPDX-License-Identifier: Apache-2.0
| For details check: Apache-2.0_

.. _Apache-2.0: https://www.apache.org/licenses/LICENSE-2.0

.. </legal notes>



*)

{attribute 'reflection'}
FUNCTION_BLOCK INTERNAL Windows125xStringPointerAssertions EXTENDS AbstractStringPointerAssertions IMPLEMENTS IWindows125xStringPointerAssertions

(*

## Short summary
This abstract property returns the class name of the concrete object, 
It's for debugging purpose

.. <legal notes>

legal notes
=================
| SPDX-FileCopyrightText: © 2024 ekvip automation GmbH <info@ekvip.de>
| SPDX-License-Identifier: Apache-2.0
| For details check: Apache-2.0_

.. _Apache-2.0: https://www.apache.org/licenses/LICENSE-2.0

.. </legal notes>

*)

PROPERTY className :CNM_AbstractObject.ClassName
GET
className := 'CNM_Assertor.Windows125xStringPointerAssertions';
END_GET
END_PROPERTY

(*

## Short summary
This assertion method checks if the current string ``stringToCheck`` contains the search string ``searchString``.
Processed strings must be in Windows-1252 or Windows-1251 encoding

**Attention:** 
	All strings are handled as null-terminated byte streams

.. <legal notes>

legal notes
=================
| SPDX-FileCopyrightText: © 2024 ekvip automation GmbH <info@ekvip.de>
| SPDX-License-Identifier: Apache-2.0
| For details check: Apache-2.0_

.. _Apache-2.0: https://www.apache.org/licenses/LICENSE-2.0

.. </legal notes>



*)

METHOD contains
VAR_INPUT
	(* current string to check *)
	stringToCheck	:POINTER TO BYTE;
	(* string must be found in ``stringToCheck`` *)
	searchString	:POINTER TO BYTE;
	(* ``TRUE`` means ignore cases; ``FALSE`` means that cases must be equal too *)
	ignoreCases		:BOOL;
	(* message if the assertion is false *)
	message			:AssertMessage;
	(* used Single Byte Character Set (SBCS), is set in Tc2_Utilities.GLOBAL_SBCS_TABLE *)
	sbcsType 		:Tc2_Utilities.E_SBCSType := Tc2_Utilities.E_SBCSType.eSBCS_WesternEuropean;
END_VAR
VAR
	(* length of current string to check *)
	lengthStringToCheck	:UDINT;
	(* length of ``searchString`` *)
	lengthSearchString	:UDINT;
	(* difference between string length and search string length *)
	maxSearchIndex :UDINT;
	(* string address we use to compare, if it's case sensitive it's equal to ``stringToCheck`` *)
	usedStringToCheck	:POINTER TO BYTE;
	(* seacrch string address we use to compare, if it's case sensitive it's equal to ``searchString`` *)
	usedSearchString	:POINTER TO BYTE;
	(* character index for the comperation *)
	character			:UDINT;
END_VAR
lengthStringToCheck := THIS^.getStringLength(stringToCheck);
lengthSearchString := THIS^.getStringLength(searchString);

IF (
	NOT THIS^.isContainsCheckNecessary(
		stringToCheck		:= stringToCheck,
		searchString		:= searchString,
		lengthStringToCheck	:= lengthStringToCheck,
		lengthSearchString	:= lengthSearchString,
		additionalText		:= THIS^.getDebugInfo('contains'),
		message				:= message
	)
) THEN
	RETURN;
END_IF

usedStringToCheck := THIS^.getNewUpperCaseString(stringToCheck, lengthStringToCheck, ignoreCases, sbcsType := sbcsType);
usedSearchString := THIS^.getNewUpperCaseString(searchString, lengthSearchString, ignoreCases, sbcsType := sbcsType);
IF ignoreCases AND_THEN ((usedStringToCheck = 0) OR_ELSE (usedSearchString = 0)) THEN
	THIS^.assertionWasWrong(message := message, additionalText := THIS^.getDebugInfo('contains, malloc failed'));
	RETURN;
END_IF

maxSearchIndex := lengthStringToCheck - lengthSearchString;
FOR (character := 0) TO (maxSearchIndex) DO
	IF (Tc2_System.MEMCMP(
			ADR(usedStringToCheck[character]),
			usedSearchString, 
			lengthSearchString
		) = CNM_ReturnTypes.ComparationResult.EQUAL
	) THEN
		THIS^.freeMemory(usedStringToCheck, ignoreCases);
		THIS^.freeMemory(usedSearchString, ignoreCases);		
		RETURN; //assert is true
	END_IF; 
END_FOR

THIS^.assertionWasWrong(message, THIS^.getDebugInfo('contains'));
THIS^.freeMemory(usedStringToCheck, ignoreCases);
THIS^.freeMemory(usedSearchString, ignoreCases);
END_METHOD

(*

## Short summary
This assertion method checks if the current string ``stringToCheck`` doesn't contain the search string ``searchString``.
Processed strings must be in Windows-1252 or Windows-1251 encoding

**Attention:** 
	All strings are handled as null-terminated byte streams

.. <legal notes>

legal notes
=================
| SPDX-FileCopyrightText: © 2024 ekvip automation GmbH <info@ekvip.de>
| SPDX-License-Identifier: Apache-2.0
| For details check: Apache-2.0_

.. _Apache-2.0: https://www.apache.org/licenses/LICENSE-2.0

.. </legal notes>



*)

METHOD containsNo
VAR_INPUT
	(* current string to check *)
	stringToCheck	:POINTER TO BYTE;
	(* string must be found in ``stringToCheck`` *)
	searchString	:POINTER TO BYTE;
	(* ``TRUE`` means ignore cases; ``FALSE`` means that cases must be equal too *)
	ignoreCases		:BOOL;
	(* message if the assertion is false *)
	message			:AssertMessage;
	(* used Single Byte Character Set (SBCS), is set in Tc2_Utilities.GLOBAL_SBCS_TABLE *)
	sbcsType 		:Tc2_Utilities.E_SBCSType := Tc2_Utilities.E_SBCSType.eSBCS_WesternEuropean;
END_VAR
VAR
	(* length of current string to check *)
	lengthStringToCheck	:UDINT;
	(* length of ``searchString`` *)
	lengthSearchString	:UDINT;
	(* difference between string length and search string length *)
	maxSearchIndex :UDINT;
	(* string address we use to compare, if it's case sensitive it's equal to ``stringToCheck`` *)
	usedStringToCheck	:POINTER TO BYTE;
	(* seacrch string address we use to compare, if it's case sensitive it's equal to ``searchString`` *)
	usedSearchString	:POINTER TO BYTE;
	(* character index for the comperation *)
	character			:UDINT;
END_VAR
lengthStringToCheck := THIS^.getStringLength(stringToCheck);
lengthSearchString := THIS^.getStringLength(searchString);

IF (
	NOT THIS^.isContainsNoCheckNecessary(
		stringToCheck		:= stringToCheck,
		searchString		:= searchString,
		lengthStringToCheck	:= lengthStringToCheck,
		lengthSearchString	:= lengthSearchString,
		additionalText		:= THIS^.getDebugInfo('containsNo'),
		message				:= message
	)
) THEN
	RETURN;
END_IF

usedStringToCheck := THIS^.getNewUpperCaseString(stringToCheck, lengthStringToCheck, ignoreCases, sbcsType := sbcsType);
usedSearchString := THIS^.getNewUpperCaseString(searchString, lengthSearchString, ignoreCases, sbcsType := sbcsType);
maxSearchIndex := lengthStringToCheck - lengthSearchString;
FOR (character := 0) TO maxSearchIndex DO
	IF (Tc2_System.MEMCMP(
			ADR(usedStringToCheck[character]),
			usedSearchString, 
			lengthSearchString
		) = CNM_ReturnTypes.ComparationResult.EQUAL
	) THEN
		THIS^.assertionWasWrong(message, THIS^.getDebugInfo('containsNo'));
		THIS^.freeMemory(usedStringToCheck, ignoreCases);
		THIS^.freeMemory(usedSearchString, ignoreCases);		
		RETURN;
	END_IF; 
END_FOR

THIS^.freeMemory(usedStringToCheck, ignoreCases);
THIS^.freeMemory(usedSearchString, ignoreCases);
END_METHOD

(*

## Short summary
This assertion method checks if the current string ``stringToCheck`` ends with the string ``end``.
Processed strings must be in Windows-1252 or Windows-1251 encoding

**Attention:** 
	All strings are handled as null-terminated byte streams

.. <legal notes>

legal notes
=================
| SPDX-FileCopyrightText: © 2024 ekvip automation GmbH <info@ekvip.de>
| SPDX-License-Identifier: Apache-2.0
| For details check: Apache-2.0_

.. _Apache-2.0: https://www.apache.org/licenses/LICENSE-2.0

.. </legal notes>



*)

METHOD endsWith
VAR_INPUT
	(* current string to check *)
	stringToCheck	:POINTER TO BYTE;
	(* string must be the end of ``stringToCheck`` *)
	end				:POINTER TO BYTE;
	(* ``TRUE`` means ignore cases; ``FALSE`` means that cases must be equal too *)
	ignoreCases		:BOOL;
	(* ``TRUE`` means truncation of spaces on the right side of ``stringToCheck``*)
	trim		:BOOL;
	(* message if the assertion is false *)
	message			:AssertMessage;
	(* used Single Byte Character Set (SBCS), is set in Tc2_Utilities.GLOBAL_SBCS_TABLE *)
	sbcsType 		:Tc2_Utilities.E_SBCSType := Tc2_Utilities.E_SBCSType.eSBCS_WesternEuropean;
END_VAR
VAR
	(* length of current string to check *)
	lengthStringToCheck	:UDINT;
	(* length of ``end`` *)
	lengthOfEnd			:UDINT;
	(* string address we use to compare, if it's case sensitive it's equal to ``stringToCheck`` *)
	usedStringToCheck	:POINTER TO BYTE;
	(* seacrch string address we use to compare, if it's case sensitive it's equal to ``end`` *)
	usedEndString		:POINTER TO BYTE;
END_VAR
lengthStringToCheck := THIS^.getStringLength(stringToCheck);
lengthOfEnd := THIS^.getStringLength(end);

THIS^.trimRight(stringToCheck, lengthStringToCheck, trim);
THIS^.trimRight(end, lengthOfEnd, trim);

IF (
	NOT THIS^.isContainsCheckNecessary(
		stringToCheck		:= stringToCheck,
		searchString		:= end,
		lengthStringToCheck	:= lengthStringToCheck,
		lengthSearchString	:= lengthOfEnd,
		additionalText		:= THIS^.getDebugInfo('endsWith'),
		message				:= message
	)
) THEN
	RETURN;
END_IF

usedStringToCheck := THIS^.getNewUpperCaseString(stringToCheck, lengthStringToCheck, ignoreCases, sbcsType := sbcsType);
usedEndString := THIS^.getNewUpperCaseString(end, lengthOfEnd, ignoreCases, sbcsType := sbcsType);

IF (Tc2_System.MEMCMP(
		ADR(usedStringToCheck[lengthStringToCheck - lengthOfEnd]),
		usedEndString, 
		lengthOfEnd
	) <> CNM_ReturnTypes.ComparationResult.EQUAL
) THEN
	THIS^.assertionWasWrong(message, THIS^.getDebugInfo('endsWith'));
END_IF;

THIS^.freeMemory(usedStringToCheck, ignoreCases);
THIS^.freeMemory(usedEndString, ignoreCases);
END_METHOD

(*

## Short summary
This method is used to free allocated memory if needed

.. <legal notes>

legal notes
=================
| SPDX-FileCopyrightText: © 2024 ekvip automation GmbH <info@ekvip.de>
| SPDX-License-Identifier: Apache-2.0
| For details check: Apache-2.0_

.. _Apache-2.0: https://www.apache.org/licenses/LICENSE-2.0

.. </legal notes>



*)

METHOD PROTECTED freeMemory
VAR_INPUT
	(* start address of the memory to free *)
	stringAddress	:POINTER TO BYTE;
	(* ``TRUE`` means free the memory, ``FALSE`` means do not free the memory *)
	freeAllocatedMemory		:BOOL;
END_VAR
IF (freeAllocatedMemory) THEN
	__DELETE(stringAddress);
END_IF
END_METHOD

(*

## Short summary
this methods copy a string and returns the start address of new string,
all small letters are capitalized in the new string.

.. <legal notes>

legal notes
=================
| SPDX-FileCopyrightText: © 2024 ekvip automation GmbH <info@ekvip.de>
| SPDX-License-Identifier: Apache-2.0
| For details check: Apache-2.0_

.. _Apache-2.0: https://www.apache.org/licenses/LICENSE-2.0

.. </legal notes>


:return: start address of a string. 
If ``createNewUpperCaseString`` is ``TRUE`` then it's a new string

*)

METHOD PROTECTED getNewUpperCaseString :POINTER TO BYTE; 
VAR_INPUT
	(* start address of the string to copy and capitalize *)
	stringAddress				:POINTER TO BYTE;
	(* length of the string ``stringAddress`` *)
	stringLength				:UDINT;
	(* 
	``TRUE means meake a copy and capitalize it, 
	``FALSE`` means return just ``stringAddress``
	and do nothing else
	*)
	createNewUpperCaseString	:BOOL;
	(* used Single Byte Character Set (SBCS), is set in Tc2_Utilities.GLOBAL_SBCS_TABLE *)
	sbcsType 		:Tc2_Utilities.E_SBCSType := Tc2_Utilities.E_SBCSType.eSBCS_WesternEuropean;
END_VAR
IF (createNewUpperCaseString) THEN
	getNewUpperCaseString := THIS^.getStringCopy(stringAddress, stringLength);
	THIS^.upperCase(getNewUpperCaseString, stringLength, sbcsType := sbcsType);
ELSE
	getNewUpperCaseString := stringAddress;
END_IF
END_METHOD

(*

## Short summary
this methods copy a string and returns the start address of new string

.. <legal notes>

legal notes
=================
| SPDX-FileCopyrightText: © 2024 ekvip automation GmbH <info@ekvip.de>
| SPDX-License-Identifier: Apache-2.0
| For details check: Apache-2.0_

.. _Apache-2.0: https://www.apache.org/licenses/LICENSE-2.0

.. </legal notes>


:return: start address of the string copy

*)

METHOD PROTECTED getStringCopy :POINTER TO BYTE
VAR_INPUT
	(* string to copy *)
	stringAddress		:POINTER TO BYTE;
	(* length of the string *)
	stringLength		:UDINT;
END_VAR
getStringCopy := __NEW(BYTE, stringLength);
IF (getStringCopy <> 0) THEN
	Tc2_System.MEMCPY(
		destAddr := getStringCopy,
		srcAddr := stringAddress,
		n := stringLength
	);
END_IF
END_METHOD

(*

## Short summary
this methods returns the length of a null-terminated string in bytes

**Attention:** 
	All strings are handled as null-terminated byte streams.

.. <legal notes>

legal notes
=================
| SPDX-FileCopyrightText: © 2024 ekvip automation GmbH <info@ekvip.de>
| SPDX-License-Identifier: Apache-2.0
| For details check: Apache-2.0_

.. _Apache-2.0: https://www.apache.org/licenses/LICENSE-2.0

.. </legal notes>


:return: length of the string

*)

METHOD PROTECTED getStringLength :UDINT
VAR_INPUT
	(* Start address of the string for which the length is to be determined *)
	stringAddress	:POINTER TO BYTE;
END_VAR
VAR CONSTANT
	(* the end of string marker *)
	END_OF_STRING	:BYTE := 16#00;
END_VAR
getStringLength := 0;
RETURN(stringAddress = 0);

WHILE (stringAddress[getStringLength] <> END_OF_STRING) DO
	getStringLength := getStringLength + 1;
END_WHILE
END_METHOD

(*

## Short summary
this methods checks if a windows-1252 or a windows-1251 character is a whitespace character

.. <legal notes>

legal notes
=================
| SPDX-FileCopyrightText: © 2024 ekvip automation GmbH <info@ekvip.de>
| SPDX-License-Identifier: Apache-2.0
| For details check: Apache-2.0_

.. _Apache-2.0: https://www.apache.org/licenses/LICENSE-2.0

.. </legal notes>


:return: ``TRUE`` means ``character`` is whitespace,
``FALSE`` means ``character`` is no whitespace 

*)

METHOD PROTECTED isCharWhiteSpace :BOOL
VAR_INPUT
	(* character to check if it's whitespace *)
	character	:BYTE;
END_VAR
VAR CONSTANT
	SPACE			:BYTE := 16#20;
	HORIZONTAL_TAB	:BYTE := 16#09;
	LINE_FEED		:BYTE := 16#0A;
	VERTICAL_TAB	:BYTE := 16#0B;
	FROM_FEED		:BYTE := 16#0C;
	CARRIAGE_RETURN	:BYTE := 16#0D;
END_VAR
CASE character OF
HORIZONTAL_TAB .. CARRIAGE_RETURN,
SPACE:
	isCharWhiteSpace := TRUE;
ELSE
	isCharWhiteSpace := FALSE;	
END_CASE
END_METHOD

(*

## Short summary
This assertion method checks if the current string ``stringToCheck`` is equal to ``expected``.
Processed strings must be in Windows-1252 or Windows-1251 encoding

**Attention:** 
	All strings are handled as null-terminated byte streams

.. <legal notes>

legal notes
=================
| SPDX-FileCopyrightText: © 2024 ekvip automation GmbH <info@ekvip.de>
| SPDX-License-Identifier: Apache-2.0
| For details check: Apache-2.0_

.. _Apache-2.0: https://www.apache.org/licenses/LICENSE-2.0

.. </legal notes>



*)

METHOD isEqualTo
VAR_INPUT
	(* current string to check *)
	stringToCheck	:POINTER TO BYTE;
	(* ``stringToCheck`` must be equal to expected *)
	expected		:POINTER TO BYTE;
	(* ``TRUE`` means ignore cases; ``FALSE`` means that cases must be equal too *)
	ignoreCases		:BOOL;
	(* message if the assertion is false *)
	message			:AssertMessage;
	(* used Single Byte Character Set (SBCS), is set in Tc2_Utilities.GLOBAL_SBCS_TABLE *)
	sbcsType 		:Tc2_Utilities.E_SBCSType := Tc2_Utilities.E_SBCSType.eSBCS_WesternEuropean;
END_VAR
VAR
	(* length of current string to check *)
	lengthStringToCheck		:UDINT;
	(* length of ``expected`` *)
	lengthExpectedString	:UDINT;
	(* string address we use to compare, if it's case sensitive it's equal to ``stringToCheck`` *)
	usedStringToCheck		:POINTER TO BYTE;
	(* seacrch string address we use to compare, if it's case sensitive it's equal to ``expected`` *)
	usedExpectedString		:POINTER TO BYTE;
END_VAR
VAR CONSTANT
	(* length of an empty string to avoid Tc2_System.MEMCMP with length 0 *)
	EMPTY_STRING_LENGTH		:UDINT := 0;
END_VAR
lengthStringToCheck := THIS^.getStringLength(stringToCheck);
lengthExpectedString := THIS^.getStringLength(expected);

IF lengthStringToCheck <> lengthExpectedString THEN
	THIS^.assertionWasWrong(message, THIS^.getDebugInfo('isEqualTo'));
	RETURN;
ELSIF (lengthExpectedString = EMPTY_STRING_LENGTH) THEN
	RETURN;
END_IF

usedStringToCheck := THIS^.getNewUpperCaseString(stringToCheck, lengthStringToCheck, ignoreCases, sbcsType := sbcsType);
usedExpectedString := THIS^.getNewUpperCaseString(expected, lengthExpectedString, ignoreCases, sbcsType := sbcsType);

IF (Tc2_System.MEMCMP(
		usedStringToCheck,
		usedExpectedString, 
		lengthExpectedString
	) <> CNM_ReturnTypes.ComparationResult.EQUAL
) THEN
	THIS^.assertionWasWrong(message, THIS^.getDebugInfo('isEqualTo'));
END_IF;

THIS^.freeMemory(usedStringToCheck, ignoreCases);
THIS^.freeMemory(usedExpectedString, ignoreCases);
END_METHOD

(*

## Short summary
This assertion method checks if the current string ``stringToCheck`` is not equal to ``unexpected``.
Processed strings must be in Windows-1252 or Windows-1251 encoding

**Attention:** 
	All strings are handled as null-terminated byte streams

.. <legal notes>

legal notes
=================
| SPDX-FileCopyrightText: © 2024 ekvip automation GmbH <info@ekvip.de>
| SPDX-License-Identifier: Apache-2.0
| For details check: Apache-2.0_

.. _Apache-2.0: https://www.apache.org/licenses/LICENSE-2.0

.. </legal notes>



*)

METHOD isNotEqualTo
VAR_INPUT
	(* current string to check *)
	stringToCheck	:POINTER TO BYTE;
	(* ``stringToCheck`` must be not equal to expected *)
	unexpected		:POINTER TO BYTE;
	(* ``TRUE`` means ignore cases; ``FALSE`` means that cases must be equal too *)
	ignoreCases		:BOOL;
	(* message if the assertion is false *)
	message			:AssertMessage;
	(* used Single Byte Character Set (SBCS), is set in Tc2_Utilities.GLOBAL_SBCS_TABLE *)
	sbcsType 		:Tc2_Utilities.E_SBCSType := Tc2_Utilities.E_SBCSType.eSBCS_WesternEuropean;
END_VAR
VAR
	(* length of current string to check *)
	lengthStringToCheck		:UDINT;
	(* length of ``unexpected`` *)
	lengthUnexpectedString	:UDINT;
	(* string address we use to compare, if it's case sensitive it's equal to ``stringToCheck`` *)
	usedStringToCheck		:POINTER TO BYTE;
	(* seacrch string address we use to compare, if it's case sensitive it's equal to ``expected`` *)
	usedUnexpectedString	:POINTER TO BYTE;
END_VAR
VAR CONSTANT
	(* length of an empty string to avoid Tc2_System.MEMCMP with length 0 *)
	EMPTY_STRING_LENGTH		:UDINT := 0;
END_VAR
lengthStringToCheck := THIS^.getStringLength(stringToCheck);
lengthUnexpectedString := THIS^.getStringLength(unexpected);

IF lengthStringToCheck = EMPTY_STRING_LENGTH AND_THEN lengthUnexpectedString = EMPTY_STRING_LENGTH THEN
	THIS^.assertionWasWrong(message, THIS^.getDebugInfo('isNotEqualTo'));
	RETURN;
END_IF

usedStringToCheck := THIS^.getNewUpperCaseString(stringToCheck, lengthStringToCheck, ignoreCases, sbcsType := sbcsType);
usedUnexpectedString := THIS^.getNewUpperCaseString(unexpected, lengthUnexpectedString, ignoreCases, sbcsType := sbcsType);

IF ( 
	(lengthStringToCheck = lengthUnexpectedString)
	AND_THEN
	Tc2_System.MEMCMP(
		usedStringToCheck,
		usedUnexpectedString, 
		lengthUnexpectedString
	) = CNM_ReturnTypes.ComparationResult.EQUAL
) THEN
	THIS^.assertionWasWrong(message, THIS^.getDebugInfo('isNotEqualTo'));
END_IF;

THIS^.freeMemory(usedStringToCheck, ignoreCases);
THIS^.freeMemory(usedUnexpectedString, ignoreCases);
END_METHOD

(*

## Short summary
This assertion method checks if the current string ``stringToCheck`` length is between ``minLength`` and ``maxLength``.
Processed strings must be in Windows-1252 or Windows-1251 encoding

**Attention:** 
	All strings are handled as null-terminated byte streams

.. <legal notes>

legal notes
=================
| SPDX-FileCopyrightText: © 2024 ekvip automation GmbH <info@ekvip.de>
| SPDX-License-Identifier: Apache-2.0
| For details check: Apache-2.0_

.. _Apache-2.0: https://www.apache.org/licenses/LICENSE-2.0

.. </legal notes>



*)

METHOD lengthIsBetween
VAR_INPUT
	(* current string to check *)
	stringToCheck	:POINTER TO BYTE;
	(* lower limit of the string length *)
	minLength		:UDINT;
	(* upper limit of the string length *)
	maxLength		:UDINT;
	(* message if the assertion is false *)
	message			:AssertMessage;
END_VAR
VAR
	(* length of ``stringToCheck`` *)
	lengthStringToCheck	:UDINT;
END_VAR
IF minLength > maxLength THEN
	THIS^.assertionWasWrong(message, THIS^.getDebugInfo('lengthIsBetween'));
	RETURN;
END_IF

lengthStringToCheck := THIS^.getStringLength(stringToCheck);

IF lengthStringToCheck < minLength OR_ELSE lengthStringToCheck > maxLength THEN
	THIS^.assertionWasWrong(message, THIS^.getDebugInfo('lengthIsBetween'));
END_IF;
END_METHOD

(*

## Short summary
This assertion method checks if the current string ``stringToCheck`` length is equal to ``expectedLength``.
Processed strings must be in Windows-1252 or Windows-1251 encoding

**Attention:** 
	All strings are handled as null-terminated byte streams

.. <legal notes>

legal notes
=================
| SPDX-FileCopyrightText: © 2024 ekvip automation GmbH <info@ekvip.de>
| SPDX-License-Identifier: Apache-2.0
| For details check: Apache-2.0_

.. _Apache-2.0: https://www.apache.org/licenses/LICENSE-2.0

.. </legal notes>



*)

METHOD lengthIsExact
VAR_INPUT
	(* current string to check *)
	stringToCheck	:POINTER TO BYTE;
	(* expected length of ``stringToCheck`` *)
	expectedLength	:UDINT;
	(* message if the assertion is false *)
	message			:AssertMessage;
END_VAR
IF (THIS^.getStringLength(stringToCheck) <> expectedLength) THEN
	THIS^.assertionWasWrong(message, THIS^.getDebugInfo('LengthIsExact'));
END_IF
END_METHOD

(*

## Short summary
This assertion method checks if the current string ``stringToCheck`` length is equal or less than to ``maxLength``.
Processed strings must be in Windows-1252 or Windows-1251 encoding

**Attention:** 
	All strings are handled as null-terminated byte streams

.. <legal notes>

legal notes
=================
| SPDX-FileCopyrightText: © 2024 ekvip automation GmbH <info@ekvip.de>
| SPDX-License-Identifier: Apache-2.0
| For details check: Apache-2.0_

.. _Apache-2.0: https://www.apache.org/licenses/LICENSE-2.0

.. </legal notes>



*)

METHOD lengthIsMax
VAR_INPUT
	(* current string to check *)
	stringToCheck	:POINTER TO BYTE;
	(* upper limit of the length of ``stringToCheck`` *)
	maxLength		:UDINT;
	(* message if the assertion is false *)
	message			:AssertMessage;
END_VAR
IF (THIS^.getStringLength(stringToCheck) > maxLength) THEN
	THIS^.assertionWasWrong(message, THIS^.getDebugInfo('LengthIsMax'));
END_IF
END_METHOD

(*

## Short summary
This assertion method checks if the current string ``stringToCheck`` length is equal or greater than to ``minLength``.
Processed strings must be in Windows-1252 or Windows-1251 encoding

**Attention:** 
	All strings are handled as null-terminated byte streams

.. <legal notes>

legal notes
=================
| SPDX-FileCopyrightText: © 2024 ekvip automation GmbH <info@ekvip.de>
| SPDX-License-Identifier: Apache-2.0
| For details check: Apache-2.0_

.. _Apache-2.0: https://www.apache.org/licenses/LICENSE-2.0

.. </legal notes>



*)

METHOD lengthIsMin
VAR_INPUT
	(* current string to check *)
	stringToCheck	:POINTER TO BYTE;
	(* lower limit of the length of ``stringToCheck`` *)
	minLength		:UDINT;
	(* message if the assertion is false *)
	message			:AssertMessage;
END_VAR
IF (THIS^.getStringLength(stringToCheck) < minLength) THEN
	THIS^.assertionWasWrong(message, THIS^.getDebugInfo('LengthIsMin'));
END_IF
END_METHOD

(*

## Short summary
This assertion method checks if the current string ``stringToCheck`` starts with string ``start``.
Processed strings must be in Windows-1252 or Windows-1251 encoding

**Attention:** 
	All strings are handled as null-terminated byte streams

.. <legal notes>

legal notes
=================
| SPDX-FileCopyrightText: © 2024 ekvip automation GmbH <info@ekvip.de>
| SPDX-License-Identifier: Apache-2.0
| For details check: Apache-2.0_

.. _Apache-2.0: https://www.apache.org/licenses/LICENSE-2.0

.. </legal notes>



*)

METHOD startsWith
VAR_INPUT
	(* current string to check *)
	stringToCheck	:POINTER TO BYTE;
	(* expected start of ``stringToCheck`` *)
	start			:POINTER TO BYTE;
	(* ``TRUE`` means ignore cases; ``FALSE`` means that cases must be equal too *)
	ignoreCases		:BOOL;
	(* ``TRUE`` means truncation of spaces on the left side of ``stringToCheck``*)
	trim		:BOOL;
	(* message if the assertion is false *)
	message			:AssertMessage;
	(* used Single Byte Character Set (SBCS), is set in Tc2_Utilities.GLOBAL_SBCS_TABLE *)
	sbcsType 		:Tc2_Utilities.E_SBCSType := Tc2_Utilities.E_SBCSType.eSBCS_WesternEuropean;
END_VAR
VAR
	(* length of current string to check *)
	lengthStringToCheck	:UDINT;
	(* length of ``start`` *)
	lengthOfStart		:UDINT;
	(* string address we use to compare, if it's case sensitive it's equal to ``stringToCheck`` *)
	usedStringToCheck	:POINTER TO BYTE;
	(* seacrch string address we use to compare, if it's case sensitive it's equal to ``start`` *)
	usedStartString		:POINTER TO BYTE;
END_VAR
lengthStringToCheck := THIS^.getStringLength(stringToCheck);
lengthOfStart := THIS^.getStringLength(start);

THIS^.trimLeft(stringToCheck, lengthStringToCheck, trim);
THIS^.trimLeft(start, lengthOfStart, trim);

IF (
	NOT THIS^.isContainsCheckNecessary(
		stringToCheck		:= stringToCheck,
		searchString		:= start,
		lengthStringToCheck	:= lengthStringToCheck,
		lengthSearchString	:= lengthOfStart,
		additionalText		:= THIS^.getDebugInfo('startsWith'),
		message				:= message
	)
) THEN
	RETURN;
END_IF

usedStringToCheck := THIS^.getNewUpperCaseString(stringToCheck, lengthStringToCheck, ignoreCases, sbcsType := sbcsType);
usedStartString := THIS^.getNewUpperCaseString(start, lengthOfStart, ignoreCases, sbcsType := sbcsType);

IF (Tc2_System.MEMCMP(
		usedStringToCheck,
		usedStartString, 
		lengthOfStart
	) <> CNM_ReturnTypes.ComparationResult.EQUAL
) THEN
	THIS^.assertionWasWrong(message, THIS^.getDebugInfo('startsWith'));
END_IF;

THIS^.freeMemory(usedStringToCheck, ignoreCases);
THIS^.freeMemory(usedStartString, ignoreCases);
END_METHOD

(*

## Short summary
This method is used to remove the whitespace from the start of the string.
It does not really remove it, it just moves the start address and decreases
the string length

.. <legal notes>

legal notes
=================
| SPDX-FileCopyrightText: © 2024 ekvip automation GmbH <info@ekvip.de>
| SPDX-License-Identifier: Apache-2.0
| For details check: Apache-2.0_

.. _Apache-2.0: https://www.apache.org/licenses/LICENSE-2.0

.. </legal notes>



*)

METHOD PROTECTED trimLeft
VAR_IN_OUT
	(* start address of the string *)
	stringAddress	:POINTER TO BYTE;
	(* length of the string ``stringAddress`` *)
	stringLength	:UDINT;
END_VAR
VAR_INPUT
	(* ``TRUE`` means remove the whitespace, ``FALSE`` means do not remove the whitespace *)
	trimString		:BOOL;
END_VAR
VAR
	(* index of the current character *)
	character		:UDINT;
	(* counter of the whitspace characters *)
	whitespaceCount	:UDINT;
	(* highest search index in the string *)
	maxSearchIndex :UDINT;
END_VAR
RETURN (NOT trimString OR_ELSE stringAddress = 0 OR_ELSE stringLength <= 0);
maxSearchIndex := stringLength - 1;
FOR character := 0 TO maxSearchIndex DO
	IF NOT (THIS^.isCharWhiteSpace(stringAddress[character])) THEN
		EXIT;
	END_IF
	whitespaceCount := whitespaceCount + 1;
END_FOR

stringAddress := stringAddress + whitespaceCount;
stringLength := stringLength - whitespaceCount;
END_METHOD

(*

## Short summary
This method is used to remove the whitespace from the end of the string.
It does not really remove it, it just decreases the string length.

.. <legal notes>

legal notes
=================
| SPDX-FileCopyrightText: © 2024 ekvip automation GmbH <info@ekvip.de>
| SPDX-License-Identifier: Apache-2.0
| For details check: Apache-2.0_

.. _Apache-2.0: https://www.apache.org/licenses/LICENSE-2.0

.. </legal notes>



*)

METHOD PROTECTED trimRight
VAR_INPUT
	(* start address of the string *)
	stringAddress	:POINTER TO BYTE;
END_VAR
VAR_IN_OUT
	(* length of the string ``stringAddress`` *)
	stringLength	:UDINT;
END_VAR
VAR_INPUT
	(* ``TRUE`` means remove the whitespace, ``FALSE`` means do not remove the whitespace *)
	trimString		:BOOL;
END_VAR
VAR
	(* index of the current character *)
	character	:LINT;
END_VAR
RETURN(NOT trimString OR_ELSE stringAddress = 0 OR_ELSE stringLength <= 0);

character := stringLength;
WHILE(character >=0) DO
	RETURN (NOT THIS^.isCharWhiteSpace(stringAddress[character := character-1]));
	stringLength := stringLength-1;
END_WHILE
END_METHOD

(*

## Short summary
This method converts the lowercase letters in an 8 bit windows-1252 or windows-1251
string to uppercase letters.

**Attention:** 
	All strings are handled as null-terminated byte streams.

.. <legal notes>

legal notes
=================
| SPDX-FileCopyrightText: © 2024 ekvip automation GmbH <info@ekvip.de>
| SPDX-License-Identifier: Apache-2.0
| For details check: Apache-2.0_

.. _Apache-2.0: https://www.apache.org/licenses/LICENSE-2.0

.. </legal notes>



*)

METHOD PROTECTED upperCase
VAR_INPUT
	(* string to ucase *)
	stringAddress	:POINTER TO BYTE;
	(* length of the string *)
	stringLength	:UDINT;
	(* used Single Byte Character Set (SBCS), is set in Tc2_Utilities.GLOBAL_SBCS_TABLE *)
	sbcsType 		:Tc2_Utilities.E_SBCSType := Tc2_Utilities.E_SBCSType.eSBCS_WesternEuropean;
END_VAR
RETURN (stringAddress = 0);

CASE sbcsType OF
Tc2_Utilities.E_SBCSType.eSBCS_WesternEuropean:
	upperCase1252(stringAddress, stringLength);
	
Tc2_Utilities.E_SBCSType.eSBCS_CentralEuropean:
	upperCase1251(stringAddress, stringLength);
ELSE
	; // do nothing
END_CASE
END_METHOD

(*

## Short summary
This method converts the lowercase letters in an 8 bit windows-1251
string to uppercase letters.

**Attention:** 
	All strings are handled as null-terminated byte streams.

.. <legal notes>

legal notes
=================
| SPDX-FileCopyrightText: © 2024 ekvip automation GmbH <info@ekvip.de>
| SPDX-License-Identifier: Apache-2.0
| For details check: Apache-2.0_

.. _Apache-2.0: https://www.apache.org/licenses/LICENSE-2.0

.. </legal notes>



*)

METHOD PROTECTED upperCase1251
VAR_INPUT
	(* string to ucase *)
	stringAddress		:POINTER TO BYTE;
	(* length of the string *)
	stringLength		:UDINT;
END_VAR
VAR
	(* index of the current character *)
	character			:UDINT := 0;
END_VAR
VAR CONSTANT
	(* NUL: $00 *)
	END_OF_STRING							:BYTE := 16#00;
	(* a *)                             	
	LOWERCASE_A								:BYTE := 16#61;
	(* z *)                             	
	LOWERCASE_Z								:BYTE := 16#7A;	
	(* а *)
	LOWERCASE_CYRILLIC_A					:BYTE := 16#E0;
	(* я *)
	LOWERCASE_CYRILLIC_YA					:BYTE := 16#FF;
	
	(* ђ *)
	LOWERCASE_CYRILLIC_DJE					:BYTE := 16#90;
	(* љ *)
	LOWERCASE_CYRILLIC_LJE					:BYTE := 16#9A;
	(* њ *)
	LOWERCASE_CYRILLIC_NJE					:BYTE := 16#9C;	
	(* џ *)
	LOWERCASE_CYRILLIC_DZHE					:BYTE := 16#9F;
	(* ё *)
	LOWERCASE_CYRILLIC_IO					:BYTE := 16#B8;
	(* є *)
	LOWERCASE_CYRILLIC_UKRAINIAN_IE			:BYTE := 16#BA;
	(* ї *)
	LOWERCASE_CYRILLIC_YI					:BYTE := 16#BF;

	(* ў *)
	LOWERCASE_CYRILLIC_SHORT_U				:BYTE := 16#A2;
	(* i *)
	LOWERCASE_CYRILLIC_UKRAINIAN_I			:BYTE := 16#B3;
	(* ѕ *)
	LOWERCASE_CYRILLIC_DZE					:BYTE := 16#BE;
	
	(* ѓ *)
	LOWERCASE_CYRILLIC_GJE					:BYTE := 16#83;
	
	(* ґ *)
	LOWERCASE_CYRILLIC_GHE_WITH_UPTURN		:BYTE := 16#B4;
	
	(* ј *)
	LOWERCASE_CYRILLIC_JE					:BYTE := 16#19;
END_VAR
WHILE stringAddress[character] <> END_OF_STRING AND_THEN character <= stringLength DO
	CASE stringAddress[character] OF
	LOWERCASE_A..LOWERCASE_Z,
	LOWERCASE_CYRILLIC_A..LOWERCASE_CYRILLIC_YA:
		stringAddress[character] := stringAddress[character] - 16#20;
	LOWERCASE_CYRILLIC_DJE,
	LOWERCASE_CYRILLIC_LJE,
	LOWERCASE_CYRILLIC_NJE..LOWERCASE_CYRILLIC_DZHE,
	LOWERCASE_CYRILLIC_IO,
	LOWERCASE_CYRILLIC_UKRAINIAN_IE,
	LOWERCASE_CYRILLIC_YI:
		stringAddress[character] := stringAddress[character] - 16#10;
	LOWERCASE_CYRILLIC_SHORT_U,
	LOWERCASE_CYRILLIC_UKRAINIAN_I,
	LOWERCASE_CYRILLIC_DZE:
		stringAddress[character] := 16#01;
	LOWERCASE_CYRILLIC_GJE:
		stringAddress[character] := 16#02;
	LOWERCASE_CYRILLIC_GHE_WITH_UPTURN:
		stringAddress[character] := 16#0F;
	LOWERCASE_CYRILLIC_JE:
		stringAddress[character] := 16#0F;
	ELSE
		; // do nothing
	END_CASE
	
	character := character + 1;
END_WHILE
END_METHOD

(*

## Short summary
This method converts the lowercase letters in an 8 bit windows-1252 
string to uppercase letters.

**Attention:** 
	All strings are handled as null terminated byte streams.

.. <legal notes>

legal notes
=================
| SPDX-FileCopyrightText: © 2024 ekvip automation GmbH <info@ekvip.de>
| SPDX-License-Identifier: Apache-2.0
| For details check: Apache-2.0_

.. _Apache-2.0: https://www.apache.org/licenses/LICENSE-2.0

.. </legal notes>



*)

METHOD PROTECTED upperCase1252
VAR_INPUT
	(* string to ucase *)
	stringAddress		:POINTER TO BYTE;
	(* length of the string *)
	stringLength		:UDINT;
END_VAR
VAR
	(* index of the current character *)
	character			:UDINT := 0;
END_VAR
VAR CONSTANT
	(* NUL: $00 *)
	END_OF_STRING							:BYTE := 16#00;
	(* a *)                             	
	LOWERCASE_A								:BYTE := 16#61;
	(* z *)                             	
	LOWERCASE_Z								:BYTE := 16#7A;
	(* ß *)                             	
	LOWERCASE_SHARP_S						:BYTE := 16#DF;
	(* ÿ *)                             	
	LOWERCASE_Y_WITH_DIAERESIS				:BYTE := 16#FF;
	(* Ÿ *)                             	
	UPPERCASE_Y_WITH_DIAERESIS				:BYTE := 16#9F;
	(* à *)                             	
	LOWERCASE_A_WITH_GRAVE					:BYTE := 16#E0;
	(* ö *)                             	
	LOWERCASE_O_WITH_DIAERESIS				:BYTE := 16#F6;
	(* ø *)                             	
	LOWERCASE_O_WITH_SLASH					:BYTE := 16#F8;
	(* þ *)                             	
	LOWERCASE_THORN							:BYTE := 16#FE;
	(* š *)                             	
	LOWERCASE_S_WITH_CARON					:BYTE := 16#9A;
	(* œ *)                             	
	LOWERCASE_OE							:BYTE := 16#9C;
	(* ž *)                             	
	LOWERCASE_Z_WITH_CARON					:BYTE := 16#9E;
	(* difference between lowercase and uppercase except for š,œ and ž *)
	DIFFERENCE_LOWERCASE_UPPERCASE			:BYTE := 16#20;
	(* for š,œ and ž the difference between lowercase and uppercase *)
	DIFFERENCE_LOWERCASE_UPPERCASE_SPECIAL	:BYTE := 16#10;
END_VAR
WHILE stringAddress[character] <> END_OF_STRING AND_THEN character <= stringLength DO
	CASE stringAddress[character] OF
	LOWERCASE_A..LOWERCASE_Z,
	LOWERCASE_A_WITH_GRAVE..LOWERCASE_O_WITH_DIAERESIS,
	LOWERCASE_O_WITH_SLASH..LOWERCASE_THORN:
		stringAddress[character] := stringAddress[character] - DIFFERENCE_LOWERCASE_UPPERCASE;
	LOWERCASE_S_WITH_CARON,
	LOWERCASE_OE,
	LOWERCASE_Z_WITH_CARON:
		stringAddress[character] := stringAddress[character] - DIFFERENCE_LOWERCASE_UPPERCASE_SPECIAL;
	LOWERCASE_Y_WITH_DIAERESIS:
		stringAddress[character] := UPPERCASE_Y_WITH_DIAERESIS;
	LOWERCASE_SHARP_S:;//for ß do nothing, because there is no capital letter for it
	ELSE
		;
	END_CASE
	
	character := character + 1;
END_WHILE
END_METHOD

END_FUNCTION_BLOCK

// ---- Assertor/Assertions/StringAssertion/classes/AbstractStringPointerAssertions.TcPOU
(*

## Short summary
Abstract class that provides methods for checking if an assert statement with contains or contains not,
makes sense based on the string lengths.

.. <legal notes>

legal notes
=================
| SPDX-FileCopyrightText: © 2022 ekvip automation GmbH <info@ekvip.de>
| SPDX-License-Identifier: Apache-2.0
| For details check: Apache-2.0_

.. _Apache-2.0: https://www.apache.org/licenses/LICENSE-2.0

.. </legal notes>



*)

{attribute 'reflection'}
FUNCTION_BLOCK INTERNAL ABSTRACT AbstractStringPointerAssertions EXTENDS AbstractAssertion 
VAR
END_VAR

(*

## Short summary
This abstract property returns the class name of the concrete object, 
It's for debugging purpose

**Attention:** 
	For derivations: **It is necessary that this property is overridden by the concrete class**

.. <legal notes>

legal notes
=================
| SPDX-FileCopyrightText: © 2022 ekvip automation GmbH <info@ekvip.de>
| SPDX-License-Identifier: Apache-2.0
| For details check: Apache-2.0_

.. _Apache-2.0: https://www.apache.org/licenses/LICENSE-2.0

.. </legal notes>

*)

PROPERTY ABSTRACT className :CNM_AbstractObject.ClassName
GET
END_GET
END_PROPERTY

(*

## Short summary
Methods for checking if an assert statement with contains or contains not,
makes sense based on the string lengths.

.. <legal notes>

legal notes
=================
| SPDX-FileCopyrightText: © 2022 ekvip automation GmbH <info@ekvip.de>
| SPDX-License-Identifier: Apache-2.0
| For details check: Apache-2.0_

.. _Apache-2.0: https://www.apache.org/licenses/LICENSE-2.0

.. </legal notes>

=
:return: ``FLASE`` means it's not necessary 
to check the string content, ``TRUE`` means
it's necessary to check the string content
to know if the assertion is true or false

*)

METHOD PROTECTED isContainsCheckNecessary :BOOL
VAR_INPUT
	(* current string to check *)
	stringToCheck	:POINTER TO BYTE;
	(* string must be found in ``stringToCheck`` *)
	searchString		:POINTER TO BYTE;
	(* length of current string to check *)
	lengthStringToCheck	:UDINT;
	(* length of ``searchString`` *)
	lengthSearchString	:UDINT;
	(* just additional text if assert is false *)	
	additionalText		:Tc2_System.T_MaxString;
	(* message if the assertion is false *)
	message				:AssertMessage;
END_VAR
isContainsCheckNecessary := FALSE;
IF	((
		lengthSearchString > lengthStringToCheck
	) OR_ELSE (
		(stringToCheck = 0) XOR (searchString = 0)
	)
) THEN
	THIS^.assertionWasWrong(message, additionalText);
	RETURN;
ELSIF	((
		(stringToCheck = 0) AND_THEN (searchString = 0)
	) OR_ELSE (
		(lengthSearchString = 0)
	) 
) THEN
	RETURN; //assert is true
END_IF
isContainsCheckNecessary := TRUE;
END_METHOD

(*

## Short summary
Methods for checking if an assert statement with contains or contains not, 
makes sense based on the string lengths

.. <legal notes>

legal notes
=================
| SPDX-FileCopyrightText: © 2022 ekvip automation GmbH <info@ekvip.de>
| SPDX-License-Identifier: Apache-2.0
| For details check: Apache-2.0_

.. _Apache-2.0: https://www.apache.org/licenses/LICENSE-2.0

.. </legal notes>

=
:return: ``FLASE`` means it's not necessary 
to check the string content, ``TRUE`` means
it's necessary to check the string content
to know if the assertion is true or false

*)

METHOD PROTECTED isContainsNoCheckNecessary :BOOL
VAR_INPUT
	(* current string to check *)
	stringToCheck		:POINTER TO BYTE;
	(* string must be found in ``stringToCheck`` *)
	searchString		:POINTER TO BYTE;
	(* length of current string to check *)
	lengthStringToCheck	:UDINT;
	(* length of ``searchString`` *)
	lengthSearchString	:UDINT;
	(* just additional text if assert is false *)	
	additionalText		:Tc2_System.T_MaxString;
	(* message if the assertion is false *)
	message				:AssertMessage;
END_VAR
isContainsNoCheckNecessary := FALSE;
IF ((
		lengthSearchString > lengthStringToCheck
	) OR_ELSE (
		(stringToCheck = 0) XOR (searchString = 0)
	)
) THEN
	RETURN; //assert is true
ELSIF ((
		(stringToCheck = 0) AND_THEN (searchString = 0)
	) OR_ELSE (	
		lengthSearchString = 0
	)
) THEN
	THIS^.assertionWasWrong(message, additionalText);
	RETURN;
END_IF
isContainsNoCheckNecessary := TRUE;
END_METHOD

END_FUNCTION_BLOCK

// ---- Assertor/Assertions/StringAssertion/Unicode/Classes/UTF-16/Utf16StringAssertions.TcPOU
(*

## Short summary
This class provides assert statements for UTF-16 strings until 255 ``WORD`` length

.. <legal notes>

legal notes
=================
| SPDX-FileCopyrightText: © 2022 ekvip automation GmbH <info@ekvip.de>
| SPDX-License-Identifier: Apache-2.0
| For details check: Apache-2.0_

.. _Apache-2.0: https://www.apache.org/licenses/LICENSE-2.0

.. </legal notes>



*)

{attribute 'reflection'}
FUNCTION_BLOCK INTERNAL Utf16StringAssertions EXTENDS AbstractAssertion IMPLEMENTS IUtf16StringAssertions
VAR
	(* class to handle the UTF-16 string assertions *)  
	assertion	:Utf16StringPointerAssertions();
END_VAR

(*

## Short summary
This abstract property returns the class name of the concrete object, 
It's for debugging purpose

.. <legal notes>

legal notes
=================
| SPDX-FileCopyrightText: © 2022 ekvip automation GmbH <info@ekvip.de>
| SPDX-License-Identifier: Apache-2.0
| For details check: Apache-2.0_

.. _Apache-2.0: https://www.apache.org/licenses/LICENSE-2.0

.. </legal notes>

*)

PROPERTY className :CNM_AbstractObject.ClassName
GET
className := 'CNM_Assertor.Utf16StringAssertions';
END_GET
END_PROPERTY

(*

## Short summary
This assertion method for UTF-16 strings checks if the current string ``stringToCheck`` 
contains the search string ``searchString``

.. <legal notes>

legal notes
=================
| SPDX-FileCopyrightText: © 2022 ekvip automation GmbH <info@ekvip.de>
| SPDX-License-Identifier: Apache-2.0
| For details check: Apache-2.0_

.. _Apache-2.0: https://www.apache.org/licenses/LICENSE-2.0

.. </legal notes>



*)

METHOD contains
VAR_INPUT
	(* current string to check *)
	stringToCheck	:WSTRING(Tc2_System.MAX_STRING_LENGTH);
	(* string must be found in ``stringToCheck`` *)
	searchString	:WSTRING(Tc2_System.MAX_STRING_LENGTH);
	(* message if the assertion is false *)
	message			:AssertMessage;
	(* ``TRUE`` means ignore cases; ``FALSE`` means cases must be equal too *)
	ignoreCases		:BOOL := FALSE;
	(*normalize both strings for check*)
	normalizeStrings :BOOL := TRUE;
END_VAR
THIS^.assertion.contains(
	stringToCheck 	:= ADR(stringToCheck),
	searchString  	:= ADR(searchString),
	ignoreCases 	:= ignoreCases,
	message 		:= message,
	normalizeStrings := normalizeStrings
);
END_METHOD

(*

## Short summary
This assertion method for UTF-16 strings checks if the current string ``stringToCheck`` contains not the search string ``searchString``

.. <legal notes>

legal notes
=================
| SPDX-FileCopyrightText: © 2022 ekvip automation GmbH <info@ekvip.de>
| SPDX-License-Identifier: Apache-2.0
| For details check: Apache-2.0_

.. _Apache-2.0: https://www.apache.org/licenses/LICENSE-2.0

.. </legal notes>



*)

METHOD containsNo
VAR_INPUT
	(* current string to check *)
	stringToCheck	:WSTRING(Tc2_System.MAX_STRING_LENGTH);
	(* string that must not be found in ``stringToCheck`` *)
	searchString	:WSTRING(Tc2_System.MAX_STRING_LENGTH);
	(* message if the assertion is false *)
	message			:AssertMessage;
	(* ``TRUE`` means ignore cases; ``FALSE`` means cases must be equal too *)
	ignoreCases		:BOOL := FALSE;
	(*normalize both strings for check*)
	normalizeStrings :BOOL := TRUE;
END_VAR
THIS^.assertion.containsNo(
	stringToCheck 	:= ADR(stringToCheck),
	searchString  	:= ADR(searchString),
	ignoreCases 	:= ignoreCases,
	message 		:= message,
	normalizeStrings := normalizeStrings
);
END_METHOD

(*

## Short summary
This assertion method for UTF-16 strings checks if the current string ``stringToCheck`` ends with the string ``end``

**Attention:** 
	end of the string is **ALWAYS** the right side of the string 
	even for writings which written from right to left like Hebrew or Arabic

.. <legal notes>

legal notes
=================
| SPDX-FileCopyrightText: © 2022 ekvip automation GmbH <info@ekvip.de>
| SPDX-License-Identifier: Apache-2.0
| For details check: Apache-2.0_

.. _Apache-2.0: https://www.apache.org/licenses/LICENSE-2.0

.. </legal notes>



*)

METHOD endsWith
VAR_INPUT
	(* current string to check *)
	stringToCheck	:WSTRING(Tc2_System.MAX_STRING_LENGTH);
	(* expected end of ``stringToCheck`` *)
	end				:WSTRING(Tc2_System.MAX_STRING_LENGTH);
	(* message if the assertion is false *)
	message			:AssertMessage;
	(* ``TRUE`` means ignore cases; ``FALSE`` means cases must be equal too *)
	ignoreCases		:BOOL := FALSE;
	(* ``TRUE`` means truncation of white-space on the right side of ``stringToCheck``*)
	trim			:BOOL := FALSE;
	(*normalize both strings for check*)
	normalizeStrings :BOOL := TRUE;
END_VAR
THIS^.assertion.endsWith(
	stringToCheck	:= ADR(stringToCheck),
	end				:= ADR(end),
	ignoreCases		:= ignoreCases,
	trim			:= trim,
	message			:= message,
	normalizeStrings := normalizeStrings
);
END_METHOD

(*

## Short summary
This assertion method checks if the current string ``stringToCheck`` is empty

.. <legal notes>

legal notes
=================
| SPDX-FileCopyrightText: © 2022 ekvip automation GmbH <info@ekvip.de>
| SPDX-License-Identifier: Apache-2.0
| For details check: Apache-2.0_

.. _Apache-2.0: https://www.apache.org/licenses/LICENSE-2.0

.. </legal notes>



*)

METHOD isEmpty
VAR_INPUT
	(* current string to check *)
	stringToCheck	:WSTRING(Tc2_System.MAX_STRING_LENGTH);
	(* message if the assertion is false *)
	message			:AssertMessage;
END_VAR
IF (stringToCheck <> "") THEN
	THIS^.assertionWasWrong(message, THIS^.getDebugInfo('isEmpty'));
END_IF
END_METHOD

(*

## Short summary
This assertion method checks if the current string ``stringToCheck`` is equal to ``expected``

.. <legal notes>

legal notes
=================
| SPDX-FileCopyrightText: © 2022 ekvip automation GmbH <info@ekvip.de>
| SPDX-License-Identifier: Apache-2.0
| For details check: Apache-2.0_

.. _Apache-2.0: https://www.apache.org/licenses/LICENSE-2.0

.. </legal notes>



*)

METHOD isEqualTo
VAR_INPUT
	(* current string to check *)
	stringToCheck	:WSTRING(Tc2_System.MAX_STRING_LENGTH);
	(* ``stringToCheck`` must be equal to expected *)
	expected		:WSTRING(Tc2_System.MAX_STRING_LENGTH);
	(* message if the assertion is false *)
	message			:AssertMessage;
	(* ``TRUE`` means ignore cases; ``FALSE`` means cases must be equal too *)
	ignoreCases		:BOOL := FALSE;
	(*normalize both strings for check*)
	normalizeStrings :BOOL := TRUE;
END_VAR
THIS^.assertion.isEqualTo(
	stringToCheck	:= ADR(stringToCheck),
	expected		:= ADR(expected),
	ignoreCases		:= ignoreCases,
	message			:= message,
	normalizeStrings := normalizeStrings
);
END_METHOD

(*

## Short summary
This assertion method checks if the current string ``stringToCheck`` is not empty

.. <legal notes>

legal notes
=================
| SPDX-FileCopyrightText: © 2022 ekvip automation GmbH <info@ekvip.de>
| SPDX-License-Identifier: Apache-2.0
| For details check: Apache-2.0_

.. _Apache-2.0: https://www.apache.org/licenses/LICENSE-2.0

.. </legal notes>



*)

METHOD isNotEmpty
VAR_INPUT
	(* current string to check *)
	stringToCheck	:WSTRING(Tc2_System.MAX_STRING_LENGTH);
	(* message if the assertion is false *)
	message			:AssertMessage;
END_VAR
IF (stringToCheck = "") THEN
	THIS^.assertionWasWrong(message, THIS^.getDebugInfo('isNotEmpty'));
END_IF
END_METHOD

(*

## Short summary
This assertion method checks if the current string ``stringToCheck`` is not equal to ``unexpected``

.. <legal notes>

legal notes
=================
| SPDX-FileCopyrightText: © 2022 ekvip automation GmbH <info@ekvip.de>
| SPDX-License-Identifier: Apache-2.0
| For details check: Apache-2.0_

.. _Apache-2.0: https://www.apache.org/licenses/LICENSE-2.0

.. </legal notes>



*)

METHOD isNotEqualTo
VAR_INPUT
	(* current string to check *)
	stringToCheck	:WSTRING(Tc2_System.MAX_STRING_LENGTH);
	(* ``stringToCheck`` must be not equal to expected *)
	unexpected		:WSTRING(Tc2_System.MAX_STRING_LENGTH);
	(* message if the assertion is false *)
	message			:AssertMessage;
	(* ``TRUE`` means ignore cases; ``FALSE`` means cases must be equal too *)
	ignoreCases		:BOOL := FALSE;
	(*normalize both strings for check*)
	normalizeStrings :BOOL := TRUE;
END_VAR
THIS^.assertion.isNotEqualTo(
	stringToCheck	:= ADR(stringToCheck),
	unexpected		:= ADR(unexpected),
	ignoreCases		:= ignoreCases,
	message			:= message,
	normalizeStrings := normalizeStrings
);
END_METHOD

(*

## Short summary
This assertion method checks if the current string ``stringToCheck`` length
is between ``minLength`` and ``maxLength``

.. <legal notes>

legal notes
=================
| SPDX-FileCopyrightText: © 2022 ekvip automation GmbH <info@ekvip.de>
| SPDX-License-Identifier: Apache-2.0
| For details check: Apache-2.0_

.. _Apache-2.0: https://www.apache.org/licenses/LICENSE-2.0

.. </legal notes>



*)

METHOD lengthIsBetween
VAR_INPUT
	(* current string to check *)
	stringToCheck	:WSTRING(Tc2_System.MAX_STRING_LENGTH);
	(* lower limit of the string length *)
	minLength		:USINT;
	(* upper limit of the string length *)
	maxLength		:USINT;
	(* string length units of measurement *)
	stringLengthUnit	:UnicodeStringLengthUnit;
	(* message if the assertion is false *)
	message			:AssertMessage;
END_VAR
THIS^.assertion.lengthIsBetween(
	stringToCheck	:= ADR(stringToCheck),
	minLength		:= minLength,
	maxLength		:= maxLength,
	stringLengthUnit := stringLengthUnit,
	message			:= message
);
END_METHOD

(*

## Short summary
This assertion method checks if the current string ``stringToCheck`` length
is equal to ``expectedLength``

.. <legal notes>

legal notes
=================
| SPDX-FileCopyrightText: © 2022 ekvip automation GmbH <info@ekvip.de>
| SPDX-License-Identifier: Apache-2.0
| For details check: Apache-2.0_

.. _Apache-2.0: https://www.apache.org/licenses/LICENSE-2.0

.. </legal notes>



*)

METHOD lengthIsExact
VAR_INPUT
	(* current string to check *)
	stringToCheck	:WSTRING(Tc2_System.MAX_STRING_LENGTH);
	(* expected length of ``stringToCheck`` *)
	expectedLength	:USINT;
	(* string length units of measurement *)
	stringLengthUnit	:UnicodeStringLengthUnit;
	(* message if the assertion is false *)
	message			:AssertMessage;
END_VAR
THIS^.assertion.lengthIsExact(
	stringToCheck	:= ADR(stringToCheck),
	expectedLength	:= expectedLength,
	stringLengthUnit := stringLengthUnit,
	message			:= message
);
END_METHOD

(*

## Short summary
This assertion method checks if the current string ``stringToCheck`` length
is equal or less than to ``maxLength``

.. <legal notes>

legal notes
=================
| SPDX-FileCopyrightText: © 2022 ekvip automation GmbH <info@ekvip.de>
| SPDX-License-Identifier: Apache-2.0
| For details check: Apache-2.0_

.. _Apache-2.0: https://www.apache.org/licenses/LICENSE-2.0

.. </legal notes>



*)

METHOD lengthIsMax
VAR_INPUT
	(* current string to check *)
	stringToCheck	:WSTRING(Tc2_System.MAX_STRING_LENGTH);
	(* upper limit of the length of ``stringToCheck`` *)
	maxLength		:USINT;
	(* string length units of measurement *)
	stringLengthUnit	:UnicodeStringLengthUnit;
	(* message if the assertion is false *)
	message			:AssertMessage;
END_VAR
THIS^.assertion.lengthIsMax(
	stringToCheck	:= ADR(stringToCheck),
	maxLength		:= maxLength,
	stringLengthUnit := stringLengthUnit,
	message			:= message
);
END_METHOD

(*

## Short summary
This assertion method checks if the current string ``stringToCheck`` length
is equal or grater than to ``minLength``

.. <legal notes>

legal notes
=================
| SPDX-FileCopyrightText: © 2022 ekvip automation GmbH <info@ekvip.de>
| SPDX-License-Identifier: Apache-2.0
| For details check: Apache-2.0_

.. _Apache-2.0: https://www.apache.org/licenses/LICENSE-2.0

.. </legal notes>



*)

METHOD lengthIsMin
VAR_INPUT
	(* current string to check *)
	stringToCheck	:WSTRING(Tc2_System.MAX_STRING_LENGTH);
	(* lower limit of the length of ``stringToCheck`` *)
	minLength		:USINT;
	(* string length units of measurement *)
	stringLengthUnit	:UnicodeStringLengthUnit;
	(* message if the assertion is false *)
	message			:AssertMessage;
END_VAR
THIS^.assertion.lengthIsMin(
	stringToCheck	:= ADR(stringToCheck),
	minLength		:= minLength,
	stringLengthUnit := stringLengthUnit,
	message			:= message
);
END_METHOD

(*

## Short summary
This methods is the setter for the callback class if an assertion was false

.. <legal notes>

legal notes
=================
| SPDX-FileCopyrightText: © 2022 ekvip automation GmbH <info@ekvip.de>
| SPDX-License-Identifier: Apache-2.0
| For details check: Apache-2.0_

.. _Apache-2.0: https://www.apache.org/licenses/LICENSE-2.0

.. </legal notes>



*)

METHOD setCallBack
VAR_INPUT
	(* the class that must be informed if an assertion is false *)
	callBack	:IAssertCallBack;  
END_VAR
SUPER^.setCallBack(callBack);
THIS^.assertion.setCallBack(callBack);
END_METHOD

(*

## Short summary
This assertion method checks if the current string ``stringToCheck`` starts with ``start``

**Attention:** 
	start of the string is **ALWAYS** the left side of the string 
	even for writings which written from right to left like Hebrew or Arabic

.. <legal notes>

legal notes
=================
| SPDX-FileCopyrightText: © 2022 ekvip automation GmbH <info@ekvip.de>
| SPDX-License-Identifier: Apache-2.0
| For details check: Apache-2.0_

.. _Apache-2.0: https://www.apache.org/licenses/LICENSE-2.0

.. </legal notes>



*)

METHOD startsWith
VAR_INPUT
	(* current string to check *)
	stringToCheck	:WSTRING(Tc2_System.MAX_STRING_LENGTH);
	(* expected start of ``stringToCheck`` *)
	start			:WSTRING(Tc2_System.MAX_STRING_LENGTH);
	(* message if the assertion is false *)
	message			:AssertMessage;
	(* ``TRUE`` means ignore cases; ``FALSE`` means cases must be equal too *)
	ignoreCases		:BOOL := FALSE;
	(* ``TRUE`` means truncation of white-space on the left side of ``stringToCheck``*)
	trim			:BOOL := FALSE;
	(*normalize both strings for check*)
	normalizeStrings :BOOL := TRUE;
END_VAR
THIS^.assertion.startsWith(
	stringToCheck	:= ADR(stringToCheck),
	start			:= ADR(start),
	ignoreCases		:= ignoreCases,
	trim			:= trim,
	message			:= message,
	normalizeStrings := normalizeStrings
);
END_METHOD

END_FUNCTION_BLOCK

// ---- Assertor/Assertions/StringAssertion/Unicode/Classes/UTF-16/Utf16StringPointerAssertions.TcPOU
(*

## Short summary
This class provides assert statements for UTF-16 strings

**Attention:** 
	All strings are handled as null terminated word streams.
	For UTF-16 is end of the string 16#00_00

.. <legal notes>

legal notes
=================
| SPDX-FileCopyrightText: © 2022 ekvip automation GmbH <info@ekvip.de>
| SPDX-License-Identifier: Apache-2.0
| For details check: Apache-2.0_

.. _Apache-2.0: https://www.apache.org/licenses/LICENSE-2.0

.. </legal notes>



*)

{attribute 'reflection'}
FUNCTION_BLOCK INTERNAL Utf16StringPointerAssertions EXTENDS AbstractStringPointerAssertions IMPLEMENTS IUtf16StringPointerAssertions
VAR
END_VAR

(*

## Short summary
This abstract property returns the class name of the concrete object, 
It's for debugging purpose

.. <legal notes>

legal notes
=================
| SPDX-FileCopyrightText: © 2022 ekvip automation GmbH <info@ekvip.de>
| SPDX-License-Identifier: Apache-2.0
| For details check: Apache-2.0_

.. _Apache-2.0: https://www.apache.org/licenses/LICENSE-2.0

.. </legal notes>

*)

PROPERTY className :CNM_AbstractObject.ClassName
GET
className := 'CNM_Assertor.Utf16StringPointerAssertions';
END_GET
END_PROPERTY

(*

## Short summary
This assertion method for UTF-16 strings checks if the current string ``stringToCheck`` contains the search string ``searchString``

**Attention:** 
	All strings are handled as null terminated word streams.
	For UTF-16 is end of the string 16#00_00

.. <legal notes>

legal notes
=================
| SPDX-FileCopyrightText: © 2022 ekvip automation GmbH <info@ekvip.de>
| SPDX-License-Identifier: Apache-2.0
| For details check: Apache-2.0_

.. _Apache-2.0: https://www.apache.org/licenses/LICENSE-2.0

.. </legal notes>



*)
{attribute 'analysis' := '-130'}
METHOD contains
VAR_INPUT
	(* current string to check *)
	stringToCheck	:POINTER TO WORD;
	(* string must be found in ``stringToCheck`` *)
	searchString	:POINTER TO WORD;
	(* ``TRUE`` means ignore cases; ``FALSE`` means cases must be equal too *)
	ignoreCases		:BOOL;
	(* message if the assertion is false *)
	message			:AssertMessage;
	(*normalize both strings for check*)
	normalizeStrings :BOOL := TRUE;
END_VAR
VAR
	(* length of ``stringToCheck`` in characters *)
	lengthStringToCheck			:UDINT;
	(* length of ``stringToCheck`` in bytes *)
	lengthStringToCheckInByte	:UDINT;
	(* length of ``stringToCheck`` in words *)
	lengthStringToCheckInWord	:UDINT;
	(* length of ``searchString`` *)
	lengthSearchString			:UDINT;
	(* length of ``searchString`` in bytes *)
	lengthSearchStringInByte	:UDINT;
	(* length of ``searchString`` in words *)
	lengthSearchStringInWord	:UDINT;
	(* character index for the comperation *)
	codePointIndex					:UDINT;
	usedCodePointsToCheck, 
    usedSearchCodePoints, 
	normalizedUsedCodePointsToCheck,
	normalizedUsedSearchCodePoints  :POINTER TO CNM_UnicodeUtilities.UnicodeCodePoint;
	usedCodePointToCheckCount, usedSearchCodePointCount :UDINT;
	maxSearchIndex :LINT;
END_VAR
VAR CONSTANT
	(*After decomposition one codepoint can extend up to 4 codepoint*)
	NORMALIZATION_FACTOR :UDINT := 4;
END_VAR
CNM_UnicodeUtilities.GetUtf16StringLength(
	utf16StringAddress := stringToCheck,
	wordCount => lengthStringToCheckInWord
);
lengthStringToCheckInByte := 2*lengthStringToCheckInWord;
 
CNM_UnicodeUtilities.GetUtf16StringLength(
	utf16StringAddress := searchString,
	wordCount => lengthSearchStringInWord
);
lengthSearchStringInByte := 2*lengthSearchStringInWord;

RETURN (((
			NOT normalizeStrings 
		) OR_ELSE (
			lengthSearchStringInWord = 0
		)
	) AND_THEN (
		NOT THIS^.isContainsCheckNecessary(
			stringToCheck		:= stringToCheck,
			searchString		:= searchString,
			lengthStringToCheck	:= lengthStringToCheckInWord,
			lengthSearchString	:= lengthSearchStringInWord,
			additionalText		:= THIS^.getDebugInfo('utf16Contains'),
			message				:= message
		) 
	)
); 

usedCodePointsToCheck := __NEW(CNM_UnicodeUtilities.UnicodeCodePoint, (lengthStringToCheckInWord+1));
IF (usedCodePointsToCheck = 0) THEN
	THIS^.assertionWasWrong(message, THIS^.getDebugInfo('utf16Contains, malloc failed'));
	RETURN;
END_IF

usedSearchCodePoints := __NEW(CNM_UnicodeUtilities.UnicodeCodePoint, (lengthSearchStringInWord+1));
IF (usedSearchCodePoints = 0) THEN
	__DELETE(usedCodePointsToCheck);
	THIS^.assertionWasWrong(message, THIS^.getDebugInfo('utf16Contains, malloc failed'));
	RETURN;
END_IF

(* convert ``stringToCheck`` to code points *)
CNM_UnicodeUtilities.GetCodepointsFromUtf16String(
	utf16StringAddress := stringToCheck, 
	utf16StringWordCount := lengthStringToCheckInWord, 
	codepointBuffer := usedCodePointsToCheck,
	bufferSize := SIZEOF(CNM_UnicodeUtilities.UnicodeCodePoint)*(lengthStringToCheckInWord+1), 
	codePointCount => usedCodePointToCheckCount
);

(* convert ``searchString`` to code points *)
CNM_UnicodeUtilities.GetCodepointsFromUtf16String(
	utf16StringAddress 	:= searchString, 
	utf16StringWordCount := lengthSearchStringInWord, 
	codepointBuffer	:= usedSearchCodePoints,
	bufferSize :=  SIZEOF(CNM_UnicodeUtilities.UnicodeCodePoint)*(lengthSearchStringInWord+1),
	codePointCount => usedSearchCodePointCount
);


IF normalizeStrings THEN
	normalizedUsedCodePointsToCheck := __NEW(CNM_UnicodeUtilities.UnicodeCodePoint, (lengthStringToCheckInWord * NORMALIZATION_FACTOR));
	IF (normalizedUsedCodePointsToCheck = 0) THEN
		THIS^.assertionWasWrong(message, THIS^.getDebugInfo('utf16Contains, malloc failed'));
		__DELETE(usedCodePointsToCheck);
		__DELETE(usedSearchCodePoints);
		RETURN;
	END_IF
	
	normalizedUsedSearchCodePoints := __NEW(CNM_UnicodeUtilities.UnicodeCodePoint, (lengthSearchStringInWord * NORMALIZATION_FACTOR));
	IF (normalizedUsedSearchCodePoints = 0) THEN
		THIS^.assertionWasWrong(message, THIS^.getDebugInfo('utf16Contains, malloc failed'));
		__DELETE(usedCodePointsToCheck);
		__DELETE(usedSearchCodePoints);
		__DELETE(normalizedUsedCodePointsToCheck);	
		RETURN;
	END_IF

	CNM_UnicodeUtilities.NormalizeCodepointsFormD(
		codePoints := usedCodePointsToCheck,
		codePointsCount := usedCodePointToCheckCount,
		normalizedCodepoints := normalizedUsedCodePointsToCheck,
		bufferSize := (lengthStringToCheckInWord * NORMALIZATION_FACTOR) * SIZEOF(CNM_UnicodeUtilities.UnicodeCodePoint),
		normalizedCodepointsCount => usedCodePointToCheckCount
	);
	__DELETE(usedCodePointsToCheck);
	usedCodePointsToCheck := normalizedUsedCodePointsToCheck;
	
	CNM_UnicodeUtilities.NormalizeCodepointsFormD(
		codePoints := usedSearchCodePoints,
		codePointsCount := usedSearchCodePointCount,
		normalizedCodepoints := normalizedUsedSearchCodePoints,
		bufferSize := (lengthSearchStringInWord * NORMALIZATION_FACTOR) * SIZEOF(CNM_UnicodeUtilities.UnicodeCodePoint),
		normalizedCodepointsCount => usedSearchCodePointCount
	);
	__DELETE(usedSearchCodePoints);
	usedSearchCodePoints := normalizedUsedSearchCodePoints;
END_IF

